	100:															// wait till password passes
		fbSoEWritePassword.Execute			:= FALSE;
		IF NOT fbSoEWritePassword.Busy THEN
			IF NOT fbSoEWritePassword.Error THEN
				iStep							:= iStep + 10;
			ELSE 
				udiADSerrorID					:= fbSoEWritePassword.AdsErrId;
				uiSoEErrorID					:= fbSoEWritePassword.SercosErrId;
				iLastStep						:= iStep;
				iStep							:= 999;
			END_IF
		END_IF
		
	110:															// Ignore offset error (P-0-0278), channel 1	
		P_0_0278_Value						:= 1;
		fbSoEWrite_ByDriveRef.stDriveRef	:= stDriveRef;
		fbSoEWrite_ByDriveRef.stDriveRef.nDriveNo:= 0;
		fbSoEWrite_ByDriveRef.nIdn			:= P_0_IDN  + 278;		// SoE Parameters Group P-0-IDN offset
		fbSoEWrite_ByDriveRef.nElement		:= EC_SOE_ELEMENT_VALUE;// Change value of the parameter
		fbSoEWrite_ByDriveRef.pSrcBuf		:= ADR(P_0_0278_Value);
		fbSoEWrite_ByDriveRef.cbBufLen		:= SIZEOF(P_0_0278_Value);
		fbSoEWrite_ByDriveRef.bExecute		:= TRUE;
		iStep								:= iStep + 10;				
		
	120,160:														// Writing done ?		
		fbSoEWrite_ByDriveRef.bExecute		:= FALSE;
		IF NOT fbSoEWrite_ByDriveRef.bBusy THEN
			IF NOT fbSoEWrite_ByDriveRef.bError THEN
				iStep							:= iStep + 10;
			ELSE
				udiADSerrorID					:= fbSoEWrite_ByDriveRef.iAdsErrId;
				uiSoEErrorID					:= fbSoEWrite_ByDriveRef.iSercosErrId;
				iLastStep						:= iStep;
				iStep							:= 999;
			END_IF	
		END_IF
		
	130:															// reset second channel if needed
		fbSoERead_ByDriveRef.stDriveRef		:= stDriveRef;
		fbSoERead_ByDriveRef.nIdn			:= P_0_IDN  + 324;		// SoE Parameters Group P-0-IDN offset
		fbSoERead_ByDriveRef.nElement		:= EC_SOE_ELEMENT_VALUE;// Change value of the parameter
		fbSoERead_ByDriveRef.pDstBuf		:= ADR(stSoE_String);
		fbSoERead_ByDriveRef.cbBufLen		:= SIZEOF(stSoE_String);
		fbSoERead_ByDriveRef.bExecute		:= TRUE;
		iStep								:= iStep + 10;				
		
	140:															// Reading done ?	skip reseting channel 2 for AX51xx	
		fbSoERead_ByDriveRef.bExecute		:= FALSE;
		IF NOT fbSoERead_ByDriveRef.bBusy THEN
			IF NOT fbSoERead_ByDriveRef.bError THEN
				bDualChannel := STRING_TO_BYTE(MID(stSoE_String.strData, 1, 4)) = 2;		// Sprawdza nazwe AX5xxx i rozpoznaje ilosc kanalow
				IF bDualChannel THEN
					iStep						:= iStep + 10;			// reset channel 2
				ELSE
					iStep						:= iStep + 30;			// skip reseting channel 2
				END_IF
			ELSE
				udiADSerrorID					:= fbSoERead_ByDriveRef.iAdsErrId;
				uiSoEErrorID					:= fbSoERead_ByDriveRef.iSercosErrId;
				iLastStep						:= iStep;
				iStep							:= 999;
			END_IF	
		END_IF
		
	150:															// Ignore offset error (P-0-0278), channel 2
		fbSoEWrite_ByDriveRef.stDriveRef.nDriveNo:= 1;
		fbSoEWrite_ByDriveRef.bExecute		:= TRUE;
		iStep								:= iStep + 10;

	170:															// Reset Drive (S-0-0099)
		fbSoEReset.Execute					:= TRUE; 
		fbSoEReset.NetId					:= ''; 
		iStep								:= iStep + 10;
		
	180:															// Wait for drive reset (S-0-0099)
		fbSoEReset.Execute					:= FALSE;
		IF NOT fbSoEReset.Busy THEN
			IF NOT fbSoEReset.Error THEN
				iStep							:= iStep + 10;
			ELSE
				udiADSerrorID					:= fbSoEReset.AdsErrId;
				uiSoEErrorID					:= fbSoEReset.SercosErrId;
				iLastStep						:= iStep;
				iStep							:= 999;
			END_IF
		END_IF
		
	190:															// Request OP State
		fbChangeSlaveState.byReguestedState	:= EC_DEVICE_STATE_OP;
		fbChangeSlaveState.bExecute			:= TRUE;
		iStep								:= iStep+10;
	
	200:															// Wait till state changed
		fbChangeSlaveState.bExecute			:= FALSE;	
		IF NOT fbChangeSlaveState.bBusy THEN
			IF NOT fbChangeSlaveState.bError THEN
				iStep							:= iStep+10;
			ELSE
				udiErrorID						:= fbChangeSlaveState.udiErrorID;
				iLastStep						:= iStep;
				iStep 							:= 999;
			END_IF				
		END_IF
		
	210:															// Set new encoder offset	
		fbSoEAX5000SetPositionOffset.Feedback:= ePositionOffsetFeedback1;	// set to feedback 1 only
		fbSoEAX5000SetPositionOffset.Execute:= TRUE; 
		iStep								:= iStep + 10;

	220:															//	offset set already?
		fbSoEAX5000SetPositionOffset.Execute:= FALSE;
		IF NOT fbSoEAX5000SetPositionOffset.Busy THEN
			IF NOT fbSoEAX5000SetPositionOffset.Error THEN
				iStep							:= iStep + 10;
			ELSE
				udiErrorID						:= fbSoEAX5000SetPositionOffset.ErrorID;
				iLastStep						:= iStep;
				iStep							:= 999;
			END_IF
		END_IF
	
	230:															//	FB Termination
		bBusy								:= FALSE;
		iStep								:= 0;

	999:															//	ERROR State
		bBusy								:=	FALSE;
		bError								:=	TRUE;
		iStep								:=	0;
	
END_CASE

fbAdsRead();
fbChangeSlaveState();
fbSoEWritePassword(Axis:=Axis);
fbSoEAX5000SetPositionOffset(Axis:=Axis);
fbSoEReadDiagNumber(Axis:=Axis);
fbSoEReset(Axis:=Axis);
fbSoEWrite_ByDriveRef();
fbSoERead_ByDriveRef();

END_FUNCTION_BLOCK

// ---- POUs/POUsAxisOnline/AX5000/FB_ChangeEtherCATSlaveState.TcPOU
//==================================================================================================
//							Beckhoff Automation Poland
//									23.05.2018
//	Blok zmienia stan EtherCAT Slave i monitoruje flage ukonczenia
//
//	Niezbedne biblioteki: Tc2_EtherCAT
//
// 	v1.1	|| TC v 3.1.4022.16	|| - optymalizacja kodu
// 	v1.0	|| TC v 3.1.4020.32	|| - pierwsza wersja
//==================================================================================================
FUNCTION_BLOCK FB_ChangeEtherCATSlaveState
VAR_INPUT
	bExecute								: BOOL;							// Start on rising edge
	sEtherCAT_NetID							: STRING;						// EtherCAT Master NetID
	nSlaveAddr								: UINT;							// EtherCAT Drive slave port
	byReguestedState						: BYTE;							(* 	16#1- EC_DEVICE_STATE_INIT  
																				16#2- EC_DEVICE_STATE_PREOP     
																				16#3- EC_DEVICE_STATE_BOOTSTRAP     
																				16#4- EC_DEVICE_STATE_SAFEOP  
																				16#8- EC_DEVICE_STATE_OP
																				16#10- EC_DEVICE_STATE_ERROR  *)
END_VAR
VAR_OUTPUT
	byActualState							: BYTE;							(* 	16#1-EC_DEVICE_STATE_INIT  
																				16#2-EC_DEVICE_STATE_PREOP     
																				16#3-EC_DEVICE_STATE_BOOTSTRAP     
																				16#4-EC_DEVICE_STATE_SAFEOP  
																				16#8-EC_DEVICE_STATE_OP
																				16#10-EC_DEVICE_STATE_ERROR  *)
	bBusy									: BOOL;
	bDone									: BOOL;
	bError									: BOOL;
	udiErrorID								: UDINT;	
END_VAR
VAR	
	fbEcReqSlaveState						: FB_EcReqSlaveState;
	fbEcGetSlaveState						: FB_EcGetSlaveState;
	timerTON								: TON;
	rtExecute								: R_TRIG;
	iState									: INT;
	iTry									: INT;							// number of tries
END_VAR

timerTON(PT:=T#500MS);
rtExecute(CLK:=bExecute);

CASE iState OF

	0:																// Init parameters
		IF rtExecute.Q THEN
			bBusy							:= TRUE;
			bDone							:= FALSE;
			bError							:= FALSE;
			udiErrorID						:= 0;
			iTry							:= 0;
			fbEcReqSlaveState.sNetId		:= sEtherCAT_NetID; 
			fbEcGetSlaveState.sNetId		:= sEtherCAT_NetID; 
			fbEcReqSlaveState.nSlaveAddr	:= nSlaveAddr; 
			fbEcGetSlaveState.nSlaveAddr	:= nSlaveAddr;
			fbEcReqSlaveState.state			:= byReguestedState;
			fbEcReqSlaveState.bExecute		:= TRUE;
			iState							:= iState + 10;			
		END_IF
		
	10:																// State request
		fbEcReqSlaveState.bExecute			:= FALSE;
		IF NOT fbEcReqSlaveState.bBusy THEN
			IF fbEcReqSlaveState.bError THEN
				iState						:= 99;
			ELSE
				iState						:= iState + 10;
			END_IF
		END_IF

		
	20:																// Request every 0.5s
		timerTON.IN							:= TRUE;
		IF timerTON.Q THEN
			timerTON.IN						:= FALSE;
			fbEcGetSlaveState.bExecute		:= TRUE;
			iState							:= iState + 10;
		END_IF
		
	30:																// Done already?
		fbEcGetSlaveState.bExecute			:= FALSE;	
		IF NOT fbEcGetSlaveState.bBusy THEN
			IF NOT fbEcGetSlaveState.bError AND fbEcGetSlaveState.state.deviceState = fbEcReqSlaveState.state THEN
				bBusy						:= FALSE;
				bDone						:= TRUE;
				iState						:= 0;
			ELSIF iTry = 40 THEN
				iState						:= 99;
			ELSE
				iTry						:= iTry + 1;
				iState						:= iState - 10;			
			END_IF
			byActualState					:= fbEcGetSlaveState.state.deviceState;
		END_IF
		
	99:																// ERROR STATE
		bError 								:= TRUE;
		bBusy								:= FALSE;
		udiErrorID							:= fbEcReqSlaveState.nErrId + fbEcGetSlaveState.nErrId;
		iState								:= 0;
		
END_CASE

fbEcReqSlaveState();
fbEcGetSlaveState();

END_FUNCTION_BLOCK

// ---- POUs/POUsAxisOnline/AX5000/FB_MotorMonitoringAX5000.TcPOU
//==================================================================================================
//							Beckhoff Automation Poland
//									22.09.2020
//	Blok funkcyjny pozwala na monitorowanie i ograniczanie momentu oraz monitoring parametru I2T dla AX5xxx.
//	Zmienne do zlinkowania zadeklarowane są wewnątrz bloku.
//	Ograniczenie i monitorowanie momentu
//	Ograniczenie momentu podawane jest przez wejście rTorqueLimit.
//	Na wyjściu podana jest wartość surowa w %, jak i przeskalowana na A (prąd) i Nm (moment).
//	Blok zwraca wartości bieżące, przefiltrowane i maksymalne.
//	Wartości maksymalne mogą być wyzerowane za pomocą zmiennej bReset.
//	Wewnętrznie wykorzystany jest blok FB_FilterEx.
//	I2T: 	Określamy okno czasowe pomiaru
//	Biblioteki: Tc2_MC2, Tc2_MC2_Drive, Tc2_Drive, Tc2_EtherCAT
//
// 	v1.4	|| TC v 3.1.4024.10		|| dostosowany do FW 2.13
// 	v1.3	|| TC v 3.1.4022.22		|| optymalizacja kod poprawiony blad wyliczenia Torque filtered
// 	v1.2	|| TC v 3.1.4022.22		|| optymalizacja kodu
// 	v1.1	|| TC v 3.1.4022.16		|| optymalizacja kodu, poprawiona flaga initialized
//  v1.0	|| TC v 3.1.4022.16		|| bazuje na FB_TorqueMonitoringEx2, dodane wyjscia zgodne z blokiem do AX8000 
//==================================================================================================
FUNCTION_BLOCK FB_MotorMonitoringAX5000
VAR CONSTANT
	rTorqueLimitLow					: REAL 		:= 0.01;				// Low limit used for bipolar torque limit value
	rTorqueLimitHigh				: REAL		:= 100.0;				// High limit used for bipolar torque limit value
END_VAR
VAR_INPUT
	bReset							: BOOL;
	rTorqueLimit					: REAL 		:= rTorqueLimitHigh; 	// Bipolar torque limit: 0-500%, resolution 0.1%, value goes to: 16#6072 (Ch A)/ 16#6872 (Ch B)
	tI2T_Window						: TIME 		:= T#100S;				// Has to be Task time * 100 * x 
																		// x - how many probes per measurement
																		// Samples - Task: 2 ms - tI2T_Window min 200 ms (1 probe), 100 probes then 20 s
																		// Task: 10 ms - tI2T_Window min 1 s (1 probe), 100 probes then 100 s
																		// If not proper time entered then it'll be adjusted
END_VAR
VAR_OUTPUT
	bError							: BOOL; 							// Communication error
	uiAdsErrId						: UINT;								// Forwarded output FB_SoeRead
	uiSercosErrId					: UINT;								// Forwarded output FB_SoeRead
	bInitialized					: BOOL;								// TRUE - Motor data read without errors, so it's possible to calculate torqe and current values in metric units
	bWarning						: BOOL;								// Overcurrent (rCurrentF > rRatedCurrent)
	rWarningCurrent					: REAL; 							// P_0_0093_Value in [A]
	rTorquePerc						: REAL;								// [%]
	rTorquePercMax					: REAL;								// Max [%]	
	rTorque							: REAL; 							// [Nm]
	rTorqueF						: REAL;								// Filtered
	rTorqueMax						: REAL;								// Max
	rCurrent						: REAL; 							// [A]
	rCurrentF						: REAL;								// Filtered
	rCurrentMax						: REAL;								// Max
	rI2T							: REAL; 							// % nominal
	rI2TMax							: REAL;
END_VAR
VAR_IN_OUT
	Axis							: AXIS_REF;
END_VAR
VAR
//======================== Internal =============================
	rTorqueRAW						: REAL; 							// -1000 .. 1000 - RAW values the same as process image	
	rContinuousStallTorque			: REAL; 							// P_0_0070_Value [Nm]
	rContinuousStallCurrent			: REAL; 							// S_0_0111_Value [A]
	rPeakCurrent					: REAL; 							// P_0_0092_Value in [A]
	rSfTorque						: REAL; 							// A --> Nm P_0_0070_Value/S_0_0111_Value [Nm/A]
	rSfCurrent						: REAL; 							// RAW --> A (-1000..1000 --> - rPeakCurrent .. rPeakCurrent)
	bFirstCycle						: BOOL := TRUE;
	iFW_High						: INT;
	iFW_Low							: INT;
	bDriveFirmware_GE_2_10			: BOOL;								// From FW >= 2.10 - different image size
	iFWPos							: INT;
	iFWLen							: INT;
	sDriveFW						: STRING(66);
	uiBipolarTorqueLimitValue AT %Q*	: UINT; 						// Raw data, linked to Bipolar torque limit value MDT, S-0-0092
	iStep							: INT;
	wInitErrorCount					: WORD;								// Initialization error counter, if bigger then 10 then error
	arr_S_0_0030_Value				: ARRAY [1..66] OF BYTE;			// till FW 2.10 total len is 66 bytes (2 - Act len, 2 - Max len, 62 - String 
	S_0_0030_Value					: STRING(61);
	P_0_0092_Value					: DWORD;
	P_0_0093_Value					: DWORD;
	P_0_0070_Value					: DWORD;
	S_0_0111_Value					: DWORD;
//========================== I2T ================================
	bCalculateI2T					: BOOL;								// TRUE in cycle when recalculation I2T necessary
	bBufferFull						: BOOL;								// TRUE when array buffer is full
	BIndex							: BYTE;								// Task no
	tI2T_WindowOld					: TIME;								// Old time window to reinit I2T calculation if necessary
	wProbeCyclesCount				: WORD;								// No of cycles for one I2T probe
	wCyclesCount					: WORD;								// Act no of cycles for one I2T probe
	wNoOfCycles						: WORD;								// Total cycles count for I2T window
	wNoOfProbes						: WORD;								// Actual number of probes for I2T calculation
	i								: INT;								// FOR loop
	rCycleTime						: REAL;								// Task time in [ms]
	rI2T_Window						: REAL;								// Time window in [ms]
	rCurrentPom						: REAL;								// Sum of current values in probe
	rCurrentAverage					: REAL;								// Arithmetical average
	rI2T_Nominal					: REAL;								// I2T for In
	rI2T_Actual						: REAL;								// I2T for real values
	arrI2TBuffer					: ARRAY[1..100] OF REAL;			// Buffer window to calculate I2T
//========================== FBs ================================
	rtReset							: R_TRIG;							// Reset trigger
	tonWait							: TON;								// Wait timer
	fbFilterEx						: FB_FilterEx;						// Filter
	fbSoERead						: FB_SoeRead;						// FB for read SoE parameters
	fbGETCURTASKINDEX   			: GETCURTASKINDEX;					// FB to check task no
//===============================================================
END_VAR

//===== Initialization, reinitialization and reset  =============
ACT_Init_Reset();
//=================== Call triggers and timers ==================
tonWait(IN:= NOT tonWait.Q, PT:= T#1S);
//============= Read params and calculations ====================
CASE iStep OF

	0: 	// Read S_0_0030 - Manufacturer version

		fbSoERead.Idn 					:= S_0_IDN + 30;
		fbSoERead.Element				:= EC_SOE_ELEMENT_VALUE;
		fbSoERead.pDstBuf				:= ADR(arr_S_0_0030_Value);
		fbSoERead.BufLen				:= SIZEOF(arr_S_0_0030_Value);
		fbSoERead.Execute				:= TRUE;
		iStep 							:= iStep + 10;

	10: // Wait till read finish 

		IF NOT fbSoERead.Busy THEN
			fbSoERead.Execute			:= FALSE;
			IF fbSoERead.Error THEN
				wInitErrorCount 		:= wInitErrorCount + 1;
				// Count > 10 then go to error and wait for reset, if not wait in warning step
				IF wInitErrorCount > 10 THEN
					uiAdsErrId			:= fbSoERead.AdsErrId;
					uiSercosErrId		:= fbSoERead.SercosErrId;
					iStep				:= 1000;								// Error step
				ELSE
					iStep				:= 900;									// Warning step
				END_IF
			ELSE
				iStep 					:= iStep + 5;
			END_IF
		END_IF

	15: // Read Drive firmware version

		MEMCPY(ADR(S_0_0030_Value), (ADR(arr_S_0_0030_Value)+4), 62);
		iFWPos							:= FIND(S_0_0030_Value,': v') + 3;
		sDriveFW						:= DELETE(S_0_0030_Value, iFWPos -1,1);
		iFWLen							:= FIND(sDriveFW,'.');
		iFW_High						:= STRING_TO_INT(LEFT(sDriveFW, iFWLen-1));
		sDriveFW						:= DELETE(sDriveFW,iFWLen,1);
		iFWLen							:= FIND(sDriveFW,' ');
		iFW_Low							:= STRING_TO_INT(LEFT(sDriveFW, iFWLen-1));
		
		bDriveFirmware_GE_2_10 			:= iFW_High >= 2 AND iFW_Low >= 10;				// Check if firmware >= 2.10
		iStep	 						:= iStep + 5;		

	20: // Read P_0_0092 - Configured channel peak current

		fbSoERead.Idn 					:= P_0_IDN + 92;
		fbSoERead.Element				:= EC_SOE_ELEMENT_VALUE;
		fbSoERead.pDstBuf				:= ADR(P_0_0092_Value);
		fbSoERead.BufLen				:= SIZEOF(P_0_0092_Value);
		fbSoERead.Execute				:= TRUE;
		iStep 							:= iStep + 10;

	30: // Wait till read finish 

		IF NOT fbSoERead.Busy THEN
			fbSoERead.Execute			:= FALSE;
			IF fbSoERead.Error THEN
				wInitErrorCount 		:= wInitErrorCount + 1;
				// Count > 10 then go to error and wait for reset, if not wait in warning step
				IF wInitErrorCount > 10 THEN
					uiAdsErrId			:= fbSoERead.AdsErrId;
					uiSercosErrId		:= fbSoERead.SercosErrId;
					iStep				:= 1000;								// Error step
				ELSE
					iStep				:= 900;									// Warning step
				END_IF
			ELSE
				iStep 					:= iStep + 10;
			END_IF
		END_IF

	40: // Read P_0_0070 - Motor continuous stall torque

		fbSoERead.Idn 					:= P_0_IDN + 70;
		fbSoERead.Element				:= EC_SOE_ELEMENT_VALUE; 
		fbSoERead.pDstBuf				:= ADR(P_0_0070_Value);
		fbSoERead.BufLen 				:= SEL(bDriveFirmware_GE_2_10, 2, 4);		// In FW GE 2.10 size is 4
		fbSoERead.Execute				:= TRUE;
		iStep 							:= iStep + 10;

	50: // Wait till read finish 

		IF NOT fbSoERead.Busy THEN
			fbSoERead.Execute			:= FALSE;
			IF fbSoERead.Error OR P_0_0070_Value = 0 THEN						// P_0_0070_Value = 0 - probably linear motor or wrong motor data
				wInitErrorCount 		:= wInitErrorCount + 1;
				// Count > 10 then go to error and wait for reset, if not wait in warning step
				IF wInitErrorCount > 10 THEN
					uiAdsErrId			:= fbSoERead.AdsErrId;
					uiSercosErrId		:= fbSoERead.SercosErrId;
					iStep				:= 1000;								// Error step
				ELSE
					iStep				:= 900;									// Warning step
				END_IF
			ELSE
				iStep 					:= iStep + 10;
			END_IF
		END_IF

	60: // Read S_0_0111 - Motor continuous stall current

		fbSoERead.Idn 					:= S_0_IDN + 111;
		fbSoERead.Element				:= EC_SOE_ELEMENT_VALUE;
		fbSoERead.pDstBuf				:= ADR(S_0_0111_Value);
		fbSoERead.BufLen				:= SIZEOF(S_0_0111_Value);
		fbSoERead.Execute				:= TRUE;
		iStep 							:= iStep + 10;
		
	70: // Wait till read finish 

		IF NOT fbSoERead.Busy THEN
			fbSoERead.Execute			:= FALSE;
			IF fbSoERead.Error OR S_0_0111_Value = 0 THEN			// S_0_0111_Value = 0 - wrong motor data
				wInitErrorCount 		:= wInitErrorCount + 1;
				// Count > 10 then go to error and wait for reset, if not wait in warning step
				IF wInitErrorCount > 10 THEN
					uiAdsErrId			:= fbSoERead.AdsErrId;
					uiSercosErrId		:= fbSoERead.SercosErrId;
					iStep				:= 1000;								// Error step
				ELSE
					iStep				:= 900;									// Warning step
				END_IF
			ELSE
				iStep 					:= iStep + 10;
			END_IF
		END_IF

	80: // Read P_0_0093 - Configured channel current

		fbSoERead.Idn 					:= P_0_IDN + 93;
		fbSoERead.Element				:= EC_SOE_ELEMENT_VALUE;
		fbSoERead.pDstBuf				:= ADR(P_0_0093_Value);
		fbSoERead.BufLen				:= SIZEOF(P_0_0093_Value);
		fbSoERead.Execute				:= TRUE;
		iStep 							:= iStep + 10;
	
	90: // Wait till read finish 

		IF NOT fbSoERead.Busy THEN
			fbSoERead.Execute			:= FALSE;
			IF fbSoERead.Error THEN
				wInitErrorCount 		:= wInitErrorCount + 1;
				// Count > 10 then go to error and wait for reset, if not wait in warning step
				IF wInitErrorCount > 10 THEN
					uiAdsErrId			:= fbSoERead.AdsErrId;
					uiSercosErrId		:= fbSoERead.SercosErrId;
					iStep				:= 1000;								// Error step
				ELSE
					iStep				:= 900;									// Warning step
				END_IF
			ELSE
				iStep 					:= iStep + 10;							
			END_IF
		END_IF
		
	100: // Read data from unit finished - we can calculate params

		rPeakCurrent 					:= DWORD_TO_REAL(P_0_0092_Value) / 1000.0;		// In [A]
		rSfCurrent 						:= rPeakCurrent / 1000.0;						// iTorque -1000..1000 --> - rPeakCurrent .. rPeakCurrent
		rContinuousStallTorque 			:= DWORD_TO_REAL(P_0_0070_Value) / 100;
		rContinuousStallCurrent 		:= DWORD_TO_REAL(S_0_0111_Value) / 1000;
		IF rContinuousStallCurrent <> 0 THEN
			rSfTorque	 				:= rContinuousStallTorque / rContinuousStallCurrent;
		END_IF
		rWarningCurrent 				:= DWORD_TO_REAL(P_0_0093_Value) / 1000;
		iStep 							:= 200;

	200: // Read cycle time - we need it for I2T calculations

		fbGETCURTASKINDEX(index => BIndex);
		IF BIndex <> 0 THEN
			iStep						:= iStep + 10;
		END_IF

	210:

		rCycleTime 						:= UDINT_TO_REAL(_TaskInfo[BIndex].CycleTime) / 10000.0;	// Scale to [ms]
		rI2T_Window 					:= TIME_TO_REAL(tI2T_Window);
		wNoOfCycles						:= REAL_TO_WORD(rI2T_Window / rCycleTime);
		// Time window too short
		IF wNoOfCycles < 100 THEN
			iStep						:= 1000;								// Error step
		ELSE
			wProbeCyclesCount 			:= wNoOfCycles / 100;
			iStep						:= 300;
		END_IF

	300: // Calculations	

		ACT_I2T();
	
	900: // Warning - wait and repeat read - problem during read motor data, i.e. EtherCAT doesn't work yet

		IF tonWait.Q THEN
			iStep 						:= 0;	// Repeat initialization phase 
		END_IF
		
	1000: // Error - wait for reset 
		;

END_CASE
//===============================================================

bError		 							:= iStep = 1000;
bInitialized 							:= iStep >= 300 AND NOT bError;
ACT_Calculations();

//========================= Warning =============================
bWarning								:= rCurrentF > rWarningCurrent;

//===================== Limit output torque =====================
IF rTorqueLimit < rTorqueLimitLow THEN
	uiBipolarTorqueLimitValue 			:= REAL_TO_UINT(rTorqueLimitHigh);			// Secure against 0 value - probably empty var connected to input
ELSE
	uiBipolarTorqueLimitValue 			:= REAL_TO_UINT(LIMIT(rTorqueLimitLow,rTorqueLimit,rTorqueLimitHigh)) * 10;
END_IF

//====================== Call SoE read FB =======================
fbSoERead(	NetId:= '',
			Timeout:= T#1s,
			Axis:= Axis);

ACTION ACT_Calculations:
//============== Raw values - always avaliable ==================
rTorquePerc								:= LREAL_TO_REAL(Axis.NcToPlc.ActTorque); 		// [%]
rTorqueRAW 								:= rTorquePerc * 10;							// -1000 .. 1000 - RAW values the same as process image
//===================== Filter current value ====================
fbFilterEx(rIn:= rTorqueRAW, tTimeConstant:= T#1S);

// Calculations	- possible only with params
IF bInitialized THEN
	rCurrent 							:= rTorqueRAW * rSfCurrent;
	rTorque 							:= rCurrent * rSfTorque;
	rCurrentF 							:= fbFilterEx.rOut * rSfCurrent;
	rTorqueF 							:= rCurrentF * rSfTorque;
END_IF

//=============== Save torque and current max values ===============
IF ABS(rCurrentMax) < ABS(rCurrentF) THEN
	rTorquePercMax						:= rTorquePerc;
	rCurrentMax 						:= rCurrentF;
	rTorqueMax 							:= rTorqueF;
END_IF
END_ACTION

ACTION ACT_I2T:
//======================= One probe =============================
rCurrentPom 							:= rCurrentPom + ABS(rCurrent);
wCyclesCount							:= wCyclesCount + 1;
bCalculateI2T							:= FALSE;
IF wCyclesCount = wProbeCyclesCount THEN
	rCurrentAverage 					:= rCurrentPom / WORD_TO_REAL(wProbeCyclesCount);
	rCurrentPom							:= 0;
	wCyclesCount						:= 0;
	bCalculateI2T						:= TRUE;							
ELSIF wCyclesCount > wProbeCyclesCount THEN
	iStep 								:= 1000;
END_IF
//===============================================================

//==================== Recalculate I2T ==========================
IF bCalculateI2T THEN
	wNoOfProbes 						:= wNoOfProbes + 1;
	bBufferFull 						:= wNoOfProbes >= 100;
	MEMMOVE(ADR(arrI2TBuffer) + 4, ADR(arrI2TBuffer), SIZEOF(arrI2TBuffer) - 4);
	arrI2TBuffer[1]						:= rCurrentAverage;
	IF bBufferFull THEN
		rI2T_Nominal					:= 100.0 * rContinuousStallCurrent;
		rI2T_Actual						:= 0;
		FOR i := 1 TO 100 DO
			rI2T_Actual					:= rI2T_Actual + arrI2TBuffer[i];
		END_FOR
	ELSE
		rI2T_Nominal					:= wNoOfProbes * rContinuousStallCurrent;
		rI2T_Actual						:= rI2T_Actual + rCurrentAverage;
	END_IF
	rI2T								:= rI2T_Actual * 100 / rI2T_Nominal; // In [%]
//====================== Save I2T max value =====================
	IF rI2TMax < rI2T THEN
		rI2TMax							:= rI2T;
	END_IF
END_IF
//===============================================================
END_ACTION

ACTION ACT_Init_Reset:
//============== Reset max values and FB ========================
rtReset(CLK:= bReset);
// Reset I2T calculations when time window changed or reset CMD
IF rtReset.Q OR tI2T_Window <> tI2T_WindowOld THEN
	BIndex								:= 0;
	wProbeCyclesCount					:= 0;
	wCyclesCount						:= 0;
	wNoOfCycles							:= 0;
	wNoOfProbes							:= 0;
	i									:= 0;
	rCycleTime							:= 0;
	rI2T_Window							:= 0;
	rCurrentPom							:= 0;
	rCurrentAverage						:= 0;
	rI2T_Nominal						:= 0;
	rI2T_Actual							:= 0;
	rI2T								:= 0;
	rI2TMax								:= 0;
	MEMSET(ADR(arrI2TBuffer), 0, SIZEOF(arrI2TBuffer));
	bBufferFull							:= FALSE;
	bCalculateI2T						:= FALSE;
	// If there is no Error then recalculate time-dipendent variables
	IF NOT bError THEN
		iStep							:= 200;
	END_IF
	tI2T_WindowOld 						:= tI2T_Window;
END_IF

IF rtReset.Q OR bFirstCycle THEN
	fbSoERead.Execute					:= FALSE;
	bWarning	 						:= FALSE;
	bDriveFirmware_GE_2_10 				:= FALSE;
	uiAdsErrId		 					:= 0;
	uiSercosErrId	 					:= 0;
	rWarningCurrent 					:= 0;
	rTorquePerc 						:= 0;
	rTorquePercMax 						:= 0;
	rTorque 							:= 0;
	rTorqueF 							:= 0;
	rTorqueMax 							:= 0;
	rCurrent 							:= 0;
	rCurrentF 							:= 0;
	rCurrentMax 						:= 0;
	rTorqueRAW 							:= 0;
	rContinuousStallTorque 				:= 0;
	rContinuousStallCurrent 			:= 0;
	rPeakCurrent 						:= 0;
	rSfTorque 							:= 0;
	rSfCurrent							:= 0;
	iStep								:= 0;
	wInitErrorCount						:= 0;
	MEMSET(ADR(arr_S_0_0030_Value), 0, SIZEOF(arr_S_0_0030_Value));
	S_0_0030_Value						:= '';
	P_0_0092_Value						:= 0;
	P_0_0093_Value						:= 0;
	P_0_0070_Value						:= 0;
	S_0_0111_Value						:= 0;
	bFirstCycle	 						:= FALSE;
END_IF
END_ACTION

END_FUNCTION_BLOCK

// ---- POUs/POUsAxisOnline/AX5000/FB_AxisDiag.TcPOU
//==================================================================================================
//							Beckhoff Automation Poland
//								23.05.2018
//					Blok do diagnostyki osi
// 	v1.1	|| TC v 3.1.4022.16	|| - optymalizacja kodu
// 	v1.0	|| TC v 3.1.4020.0	|| - pierwsza wersja
//==================================================================================================
FUNCTION_BLOCK FB_AxisDiag
VAR_INPUT
	IPCNetID							: T_AmsNetId; 	(* AmsNetId of the IPC *)
	Timeout								: TIME := DEFAULT_ADS_TIMEOUT;
	Reset								: BOOL;
	GetDiag								: BOOL;
END_VAR
VAR_IN_OUT
	Axis	 							: AXIS_REF;
	stAX5000Diag						: ST_AX5000Diag;
END_VAR
VAR_OUTPUT
	Error								: BOOL;
	AdsErrId							: UINT;
	SercosErrId							: UINT;
	ResetAct							: BOOL;
	DiagAct								: BOOL;
	Busy								: BOOL;
END_VAR
VAR
	iState								: INT;
	iSubState							: INT;
	GetDriveRef							: BOOL;
	DriveRef								: ST_DriveRef; (* contains sNetID of EcMaster, nSlaveAddr of EcDrive, nDriveNo of EcDrive, either preset or read from NC *)
	AxisID								: UDINT;

	C1DErrorPrev							: BOOL;
	WcStateErrorPrev						: BOOL;
	AxisErrorPrev							: BOOL;
	OperationalPrev						: BOOL;
	ResetPrev							: BOOL;
	GetDiagPrev							: BOOL;

	fbSoERead							: FB_SoERead;
	fbDiagMessage 						: FB_SoEReadDiagMessage;
	fbClassXDiag							: FB_SoEReadClassXDiag;
	fbDiagNumber						: FB_SoEReadDiagNumber;
	fbDiagNumberList						: FB_SoEReadDiagNumberList;

	fbReset								: FB_SoEReset;
	fbDelay								: TON;
	fbGetSlaveState 						: FB_EcGetSlaveState;
	fbReqSlaveState 						: FB_EcReqSlaveState;
	fbNcReset 							: MC_Reset;

	fbAdsRead							: ADSREAD;
	readBuffer							: ARRAY[0..9] OF BYTE;
	Ids									: T_AmsNetIdArr;
	strSoEString							: ST_SoE_String;
END_VAR
VAR CONSTANT
	NCIDXG_AXPARMS					: UDINT := 16#00004000;	(* Axis with ID: Parameter 			*)
	NCIDXO_AXP_HWAMSADDR			: UDINT := 16#00000031;
END_VAR

stAX5000Diag.bOperational	:= Axis.NcToPlc.StateDWord.0;
stAX5000Diag.bC1DError	 	:= Axis.NcToPlc.StateDWord.28;
stAX5000Diag.bWcStateError 	:= Axis.NcToPlc.StateDWord.30;
stAX5000Diag.bAxisError		:= Axis.NcToPlc.StateDWord.31;
stAX5000Diag.iAxisErrorCode	:= Axis.NcToPlc.ErrorCode;

CASE iState OF
0:	(* idle *)
	GetDriveRef 	:= (DriveRef.nSlaveAddr = 0);

	IF GetDriveRef THEN
		Busy			:= TRUE;
		Error			:= FALSE;
		AdsErrId		:= 0;
		SercosErrId		:= 0;
		iState 			:= 1;
		iSubState		:= 0;
		AxisID 			:= Axis.NcToPlc.AxisId;

	ELSIF Reset AND NOT ResetPrev THEN
		Busy			:= TRUE;
		ResetAct		:= TRUE;
		ResetPrev		:= Reset;
		Error			:= FALSE;
		AdsErrId		:= 0;
		SercosErrId		:= 0;
		iState 			:= 2;
		iSubState		:= 0;
		AxisID 			:= Axis.NcToPlc.AxisId;

	ELSIF GetDiag AND NOT GetDiagPrev OR
		(stAX5000Diag.bC1DError AND NOT C1DErrorPrev) OR (NOT stAX5000Diag.bC1DError AND C1DErrorPrev) (* rising/falling C1D *) OR
		(stAX5000Diag.bWcStateError AND NOT WcStateErrorPrev) OR (NOT stAX5000Diag.bWcStateError AND WcStateErrorPrev) (* rising/falling WcState *) OR
		(stAX5000Diag.bAxisError AND NOT AxisErrorPrev) OR (NOT stAX5000Diag.bAxisError AND AxisErrorPrev) (* rising/falling NcError *) OR
		(stAX5000Diag.bOperational AND NOT OperationalPrev) OR (NOT stAX5000Diag.bOperational AND OperationalPrev) (* rising/falling Enable *) THEN

		Busy			:= TRUE;
		DiagAct			:= TRUE;
		GetDiagPrev		:= GetDiag;
		Error			:= FALSE;
		AdsErrId		:= 0;
		SercosErrId		:= 0;
		iState 			:= 3;
		iSubState		:= 0;
		AxisID 			:= Axis.NcToPlc.AxisId;

		(* set/clear flags *)
		C1DErrorPrev		:= stAX5000Diag.bC1DError;
		WcStateErrorPrev	:= stAX5000Diag.bWcStateError;
		AxisErrorPrev		:= stAX5000Diag.bAxisError;
		OperationalPrev		:= stAX5000Diag.bOperational;

	ELSE
		ResetAct	:= FALSE;
		DiagAct		:= FALSE;
	END_IF

1:	(* get drive reference *)
	M_GetDriveRef();

2:	(* reset and state change *)
	M_Reset();

3:	(* get diag data *)
	M_GetDiagnosis();

END_CASE

(* clear latch *)
ResetPrev	:= ResetPrev AND Reset;
GetDiagPrev	:= GetDiagPrev AND GetDiag;

ACTION M_GetDiagnosis:
CASE iSubState OF
0:	fbClassXDiag(
		NetId		:= IPCNetID,
		Execute		:= TRUE,
		DiagClass 	:= 1,
		Timeout		:= DEFAULT_ADS_TIMEOUT,
		Axis		:= Axis,
	);

	IF NOT fbClassXDiag.Busy THEN
		fbClassXDiag(Execute:= FALSE,Axis := Axis);

		IF NOT fbClassXDiag.Error THEN
			stAX5000Diag.wClass1Diag	:= fbClassXDiag.ClassXDiag;
			stAX5000Diag.stClass1Diag	:= F_ConvWordToSTAX5000C1D(stAX5000Diag.wClass1Diag);
		ELSE
			Error			:= TRUE;
			AdsErrId		:= fbClassXDiag.AdsErrId;
			SercosErrId	:= fbClassXDiag.SercosErrId;
		END_IF
		iSubState	:= iSubState + 1;
	END_IF

1:	fbDiagMessage(
		NetId	:= IPCNetID,
		Execute	:= TRUE,
		Timeout	:= DEFAULT_ADS_TIMEOUT,
		Axis	:= Axis,
	);

	IF NOT fbDiagMessage.Busy THEN
		fbDiagMessage(Execute:= FALSE,Axis := Axis);

		IF NOT fbDiagMessage.Error THEN
			stAX5000Diag.strDiagMessage := LEFT(fbDiagMessage.DiagMessage.strData, UINT_TO_INT(fbDiagMessage.DiagMessage.iActualSize));
		ELSE
			Error			:= TRUE;
			AdsErrId		:= fbDiagMessage.AdsErrId;
			SercosErrId	:= fbDiagMessage.SercosErrId;
		END_IF
		iSubState	:= iSubState + 1;
	END_IF

2:	fbDiagNumber(
		NetId	:= IPCNetID,
		Execute	:= TRUE,
		Timeout	:= DEFAULT_ADS_TIMEOUT,
		Axis	:= Axis,
	);

	IF NOT fbDiagNumber.Busy THEN
		fbDiagNumber(Execute:= FALSE,Axis := Axis);

		IF NOT fbDiagNumber.Error THEN
			stAX5000Diag.iDiagNumber := fbDiagNumber.DiagNumber;
		ELSE
			Error			:= TRUE;
			AdsErrId		:= fbDiagNumber.AdsErrId;
			SercosErrId	:= fbDiagNumber.SercosErrId;
		END_IF
		iSubState	:= iSubState + 1;
	END_IF

3:	fbSoERead(
		NetId	:= IPCNetID,
		Execute	:= TRUE,
		Idn		:= 135,
		Element	:=16#44,
		pDstBuf	:=ADR(stAX5000Diag.wDriveStatus),
		BufLen	:=SIZEOF(stAX5000Diag.wDriveStatus),
		Timeout	:= DEFAULT_ADS_TIMEOUT,
		Axis	:= Axis,
	);

	IF NOT fbSoERead.Busy THEN
		fbSoERead(Execute:= FALSE,Axis := Axis);
		IF NOT fbSoERead.Error THEN
			stAX5000Diag.stDriveStatus := F_ConvWordToSTAX5000DriveStatus(stAX5000Diag.wDriveStatus);
			iSubState		:= iSubState + 1;
		ELSE
			Error			:= TRUE;
			AdsErrId		:= fbSoERead.AdsErrId;
			SercosErrId	:= fbSoERead.SercosErrId;
			iSubState		:= iSubState + 2;
		END_IF
	END_IF

4:	fbSoERead(
		NetId	:= IPCNetID,
		Execute	:= TRUE,
		Idn		:= stAX5000Diag.stDriveStatus.iActOpModeParNum,
		Element	:=16#44,
		pDstBuf	:=ADR(stAX5000Diag.stDriveStatus.eActOpMode),
		BufLen	:=SIZEOF(stAX5000Diag.stDriveStatus.eActOpMode),
		Timeout	:= DEFAULT_ADS_TIMEOUT,
		Axis	:= Axis,
	);

	IF NOT fbSoERead.Busy THEN
		fbSoERead(Execute:= FALSE,Axis := Axis);
		IF NOT fbSoERead.Error THEN
			;
		ELSE
			Error			:= TRUE;
			AdsErrId		:= fbSoERead.AdsErrId;
			SercosErrId	:= fbSoERead.SercosErrId;
		END_IF
		iSubState	:= iSubState + 1;
	END_IF

5:	fbGetSlaveState(
		sNetId		:= DriveRef.sNetId,
		nSlaveAddr	:= DriveRef.nSlaveAddr,
		bExecute	:= TRUE,
		tTimeout	:= DEFAULT_ADS_TIMEOUT,
	);

	IF NOT fbGetSlaveState.bBusy THEN
		fbGetSlaveState(bExecute:= FALSE);
		IF NOT fbGetSlaveState.bError THEN
			stAX5000Diag.stEcSlaveState := fbGetSlaveState.state;
			stAX5000Diag.stEcSlaveStateBits := F_ConvSlaveStateToBits(fbGetSlaveState.state);
		ELSE
			Error			:= TRUE;
			AdsErrId		:= UDINT_TO_UINT(fbGetSlaveState.nErrId);
		END_IF

		IF stAX5000Diag.stEcSlaveStateBits.bError THEN
			IF stAX5000Diag.stEcSlaveStateBits.bPreop THEN
				(* read S21 - IDN List of Invalid operation data for CP2 (Preop->SaveOp) *)
				MEMSET(ADR(stAX5000Diag.stCPxInvParamList), 0, SIZEOF(stAX5000Diag.stCPxInvParamList));
				stAX5000Diag.bPreopToSafeOpError := TRUE;
				stAX5000Diag.bSafeOpToOpError := FALSE;
				iSubState	:= iSubState + 1;
			ELSIF stAX5000Diag.stEcSlaveStateBits.bSafeOp THEN
				(* read S22 - IDN List of Invalid operation data for CP3 (SaveOp->Op) *)
				MEMSET(ADR(stAX5000Diag.stCPxInvParamList), 0, SIZEOF(stAX5000Diag.stCPxInvParamList));
				stAX5000Diag.bPreopToSafeOpError := FALSE;
				stAX5000Diag.bSafeOpToOpError := TRUE;
				iSubState	:= iSubState + 2;
			ELSE
				(* Skip S21 + S22 *)
				MEMSET(ADR(stAX5000Diag.stCPxInvParamList), 0, SIZEOF(stAX5000Diag.stCPxInvParamList));
				stAX5000Diag.bPreopToSafeOpError := FALSE;
				stAX5000Diag.bSafeOpToOpError := FALSE;
				iSubState	:= iSubState + 3;
			END_IF
		ELSE
			(* Skip S21 + S22 *)
			MEMSET(ADR(stAX5000Diag.stCPxInvParamList), 0, SIZEOF(stAX5000Diag.stCPxInvParamList));
			stAX5000Diag.bPreopToSafeOpError := FALSE;
			stAX5000Diag.bSafeOpToOpError := FALSE;
			iSubState	:= iSubState + 3;
		END_IF
	END_IF

6:	(* read S21 - IDN List of Invalid operation data for CP2 (Preop->SaveOp) *)
	fbSoERead(
		NetId	:= IPCNetID,
		Execute	:= TRUE,
		Idn		:= 21,
		Element	:=16#40,
		pDstBuf	:=ADR(stAX5000Diag.stCPxInvParamList),
		BufLen	:=SIZEOF(stAX5000Diag.stCPxInvParamList),
		Timeout	:= DEFAULT_ADS_TIMEOUT,
		Axis	:= Axis,
	);

	IF NOT fbSoERead.Busy THEN
		fbSoERead(Execute:= FALSE,Axis := Axis);
		IF NOT fbSoERead.Error THEN
			;
		ELSE
			Error			:= TRUE;
			AdsErrId		:= fbSoERead.AdsErrId;
			SercosErrId	:= fbSoERead.SercosErrId;
		END_IF
		iSubState	:= iSubState + 2;
	END_IF

7:	(* read S22 - IDN List of Invalid operation data for CP3 (SaveOp->Op) *)
	fbSoERead(
		NetId	:= IPCNetID,
		Execute	:= TRUE,
		Idn		:= 22,
		Element	:=16#40,
		pDstBuf	:=ADR(stAX5000Diag.stCPxInvParamList),
		BufLen	:=SIZEOF(stAX5000Diag.stCPxInvParamList),
		Timeout	:= DEFAULT_ADS_TIMEOUT,
		Axis	:= Axis,
	);

	IF NOT fbSoERead.Busy THEN
		fbSoERead(Execute:= FALSE,Axis := Axis);
		IF NOT fbSoERead.Error THEN
			;
		ELSE
			Error			:= TRUE;
			AdsErrId		:= fbSoERead.AdsErrId;
			SercosErrId	:= fbSoERead.SercosErrId;
		END_IF
		iSubState	:= iSubState + 1;
	END_IF

8:	fbDiagNumberList(
		NetId			:= IPCNetID,
		Execute			:= TRUE,
		Timeout			:= DEFAULT_ADS_TIMEOUT,
		pDiagNumber		:= ADR(stAX5000Diag.stDiagNumberList),
		Size			:= SIZEOF(stAX5000Diag.stDiagNumberList),
		Axis			:= Axis,
	);

	IF NOT fbDiagNumberList.Busy THEN
		fbDiagNumberList(Execute:= FALSE,Axis := Axis);

		IF fbDiagNumberList.Error THEN
			Error			:= TRUE;
			AdsErrId		:= fbDiagNumberList.AdsErrId;
			SercosErrId	:= fbDiagNumberList.SercosErrId;
		END_IF

		IF (stAX5000Diag.strMotorType = '') OR (stAX5000Diag.strDriveType = '') THEN
			iSubState	:= iSubState + 1;
		ELSE
			DiagAct	:= FALSE;
			iSubState	:= 0;
			iState		:= 0;
			Busy		:= FALSE;
		END_IF
	END_IF

9:	fbSoERead(
		NetId	:= IPCNetID,
		Execute	:= TRUE,
		Idn		:= P_0_IDN + 53,
		Element	:=16#44,
		pDstBuf	:=ADR(strSoEString),
		BufLen	:=SIZEOF(strSoEString),
		Timeout	:= DEFAULT_ADS_TIMEOUT,
		Axis	:= Axis,
	);

	IF NOT fbSoERead.Busy THEN
		fbSoERead(Execute:= FALSE,Axis := Axis);
		IF NOT fbSoERead.Error THEN
			MEMSET(ADR(stAX5000Diag.strMotorType),0,SIZEOF(stAX5000Diag.strMotorType));
			MEMCPY(ADR(stAX5000Diag.strMotorType),ADR(strSoEString.strData),MIN(SIZEOF(stAX5000Diag.strMotorType),strSoEString.iActualSize));
		ELSE
			Error			:= TRUE;
			AdsErrId		:= fbSoERead.AdsErrId;
			SercosErrId	:= fbSoERead.SercosErrId;
		END_IF
		iSubState	:= iSubState + 1;
	END_IF

10:	fbSoERead(
		NetId	:= IPCNetID,
		Execute	:= TRUE,
		Idn		:= P_0_IDN + 324,
		Element	:=16#44,
		pDstBuf	:=ADR(strSoEString),
		BufLen	:=SIZEOF(strSoEString),
		Timeout	:= DEFAULT_ADS_TIMEOUT,
		Axis	:= Axis,
	);

	IF NOT fbSoERead.Busy THEN
		fbSoERead(Execute:= FALSE,Axis := Axis);
		IF NOT fbSoERead.Error THEN
			MEMSET(ADR(stAX5000Diag.strDriveType),0,SIZEOF(stAX5000Diag.strDriveType));
			MEMCPY(ADR(stAX5000Diag.strDriveType),ADR(strSoEString.strData),MIN(SIZEOF(stAX5000Diag.strDriveType),strSoEString.iActualSize));
		ELSE
			Error			:= TRUE;
			AdsErrId		:= fbSoERead.AdsErrId;
			SercosErrId	:= fbSoERead.SercosErrId;
		END_IF
		DiagAct	:= FALSE;
		iSubState	:= 0;
		iState		:= 0;
		Busy		:= FALSE;
	END_IF


END_CASE
END_ACTION

ACTION M_GetDriveRef:
(* get reference from NC *)
fbAdsRead(
	NETID	:= IPCNetID,
	PORT	:= AMSPORT_R0_NC,
	IDXGRP	:= NCIDXG_AXPARMS + Axis.NcToPlc.AxisId,
	IDXOFFS	:= NCIDXO_AXP_HWAMSADDR,
	LEN		:= SIZEOF(readBuffer) ,
	DESTADDR:= ADR(readBuffer),
	READ	:= TRUE,
	TMOUT	:= Timeout
);

IF NOT fbAdsRead.BUSY THEN
	fbAdsRead(READ := FALSE);
	stAX5000Diag.nNCAxisID := Axis.NcToPlc.AxisId;

	IF NOT fbAdsRead.ERR THEN
		MEMCPY(ADR(Ids), ADR(readBuffer), SIZEOF(Ids)); 										(* readBuffer[0..5] *)
		MEMCPY(ADR(DriveRef.nSlaveAddr), ADR(readBuffer[6]), SIZEOF(DriveRef.nSlaveAddr));  	(* readBuffer[6..7] *)
		MEMCPY(ADR(DriveRef.nDriveNo), ADR(readBuffer[8]), SIZEOF(DriveRef.nDriveNo));  		(* readBuffer[8..9] *)

		(* create string out of byte array *)
		DriveRef.sNetId := F_CreateAmsNetId(Ids);
		GetDriveRef := FALSE;
	END_IF

	Busy	:= FALSE;
	iState	:= 0;
END_IF
END_ACTION

ACTION M_Reset:
CASE iSubState OF
0:
	IF stAX5000Diag.bWcStateError OR stAX5000Diag.bC1DError THEN
		(* ResetAmplifier *)
		iSubState := iSubState + 1;
	ELSIF (NOT stAX5000Diag.bOperational) OR stAX5000Diag.bAxisError OR (stAX5000Diag.iAxisErrorCode <> 0) THEN
		(* NC Reset only *)
		iSubState := 6;
	ELSE
		(* reset not required *)
		iSubState	:= 0;
		iState		:= 0;
		Busy		:= FALSE;
		ResetAct	:= FALSE;
	END_IF

1:	(* ResetAmplifier *)
	fbReset(
		NetId	:= IPCNetID,
		Execute	:= TRUE,
		Timeout	:= DEFAULT_ADS_TIMEOUT,
		Axis	:= Axis,
	);
	IF NOT fbReset.Busy THEN
		fbReset(Execute:= FALSE, Axis:= Axis);

		IF NOT fbReset.Error THEN
			iSubState	:= iSubState + 1;
		ELSE
			Error			:= TRUE;
			AdsErrId		:= fbReset.AdsErrId;
			SercosErrId		:= fbReset.SercosErrId;
			Busy			:= FALSE;
			ResetAct		:= FALSE;
			iSubState		:= 0;
			iState			:= 0;
		END_IF
	END_IF

2:	fbDelay(IN:=TRUE, PT:=t#3s);
	IF fbDelay.Q THEN
		fbDelay(IN:=FALSE);
		iSubState	:= iSubState + 1;
	END_IF

3:	fbGetSlaveState(
		sNetId		:= DriveRef.sNetId,
		nSlaveAddr	:= DriveRef.nSlaveAddr,
		bExecute	:= TRUE,
		tTimeout	:= DEFAULT_ADS_TIMEOUT,
	);

	IF NOT fbGetSlaveState.bBusy THEN
		fbGetSlaveState(bExecute:= FALSE);

		IF NOT fbGetSlaveState.bError THEN
			IF Axis.NcToPlc.StateDWord.31 OR (Axis.NcToPlc.ErrorCode <> 0) THEN
				iSubState	:= 6;
			ELSE
				Busy		:= FALSE;
				ResetAct	:= FALSE;
				iSubState	:= 0;
				iState		:= 0;
			END_IF
		ELSE
			Error			:= TRUE;
			AdsErrId		:= UDINT_TO_UINT(fbGetSlaveState.nErrId);
			Busy			:= FALSE;
			ResetAct		:= FALSE;
			iSubState		:= 0;
			iState			:= 0;
		END_IF
	END_IF

5:	(* set op *)
	fbReqSlaveState(
		sNetId		:= DriveRef.sNetId,
		nSlaveAddr	:= DriveRef.nSlaveAddr,
		bExecute	:= TRUE,
		tTimeout	:= DEFAULT_ADS_TIMEOUT,
		state		:= EC_DEVICE_STATE_OP);

	IF NOT fbReqSlaveState.bBusy THEN
		fbReqSlaveState(bExecute:= FALSE);

		IF NOT fbReqSlaveState.bError THEN
			iSubState	:= iSubState + 1;
		ELSE
			Error		:= TRUE;
			AdsErrId	:= UDINT_TO_UINT(fbReqSlaveState.nErrId);
			Busy		:= FALSE;
			ResetAct	:= FALSE;
			iSubState	:= 0;
			iState		:= 0;
		END_IF
	END_IF

6:	fbNcReset(
		Execute:= TRUE,
		Axis:= Axis,
	);
	IF fbNcReset.Done OR fbNcReset.Error THEN
		IF fbNcReset.Error THEN
			Error 		:= TRUE;
			AdsErrId 	:= UDINT_TO_UINT(fbNcReset.ErrorID);
		END_IF

		iSubState	:= 0;
		iState		:= 0;
		Busy		:= FALSE;
		ResetAct	:= FALSE;
		fbNcReset(Execute:= FALSE, Axis:= Axis);
	END_IF
END_CASE
END_ACTION

END_FUNCTION_BLOCK

// ---- POUs/POUsAxisOnline/FBs/F_AxErrMsg.TcPOU
//==================================================================================================
//							Beckhoff Automation Poland
//								7.12.2018
//		Funkcja konwertujaca nr bledu na opis
// 	v1.0	|| TC v 3.1.4022.27	|| - pierwsza wersja
//==================================================================================================
FUNCTION F_AxErrMsg : STRING(255)
VAR_INPUT
	iErrID: UDINT;
END_VAR
VAR
	sMsg: STRING(255);
END_VAR

(* these err msgs are taken straight from infosys ....
http://infosys.beckhoff.com/content/1033/tcncerrcode/html/tcncerrorcodesoverview.htm?id=27430  
*)

IF iErrID < 1 THEN
	sMsg := '';
	F_AxErrMsg := sMsg;
	RETURN;
END_IF

CASE iErrID OF
(* NC AXIS ERRORS *)
	16#4000: sMsg := '4000 internal "Internal error" Internal system error in the NC on ring 0, no further details.';
	16#4001: sMsg := '4001 memory "Memory error" The ring-0 memory management is not providing the required memory. This is usually a result of another error, as a result of which the controller will halt normal operation (now if not …';
	16#4002: sMsg := '4002 internal "Nc retain data error (persistent data)" Error while loading the Nc retain data. The axes concerned are no longer referenced (status flag "Homed" is set to FALSE).';
	16#4010: sMsg := '4010 parameter "Channel identifier not allowed" Either an unacceptable value (not 1...255) has been used, or a channel that does not exist in the system has been named.';
	16#4011: sMsg := '4011 parameter "Group identifier not allowed" Either an unacceptable value (not 1...255) has been used, or a group that does not exist in the system has been named.';
	16#4012: sMsg := '4012 parameter "Axis identifier not allowed" Either an unacceptable value (not 1...255) has been used, or an axis that does not exist in the system has been named.';
	16#4013: sMsg := '4013 parameter "Encoder identifier not allowed" Either an unacceptable value (not 1...255) has been used, or a encoder that does not exist in the system has been named.';
	16#4014: sMsg := '4014 parameter "Controller identifier not allowed" Either an unacceptable value (not 1...255) has been used, or a controller that does not exist in the system has been named.';
	16#4015: sMsg := '4015 parameter "Drive identifier not allowed" Either an unacceptable value (not 1...255) has been used, or a drive that does not exist in the system has been named.';
	16#4016: sMsg := '4016 parameter "Table identifier not allowed" Either an unacceptable value (not 1...255) has been used, or a table that does not exist in the system has been named.';
	16#4020: sMsg := '4020 internal "No process image" No PLC-axis interface during creation of an axis.';
	16#4021: sMsg := '4021 internal "No process image" No axis-PLC interface during creation of an axis.';
	16#4022: sMsg := '4022 internal "No process image" No encoder-I/O interface during creation of an axis.';
	16#4023: sMsg := '4023 internal "No process image" No I/O-encoder interface during creation of an axis.';
	16#4024: sMsg := '4024 internal "No process image" No drive-I/O interface during creation of an axis.';
	16#4025: sMsg := '4025 internal "No process image" No I/O-drive interface during creation of an axis.';
	16#4030: sMsg := '4030 internal "Coupling type not allowed" Unacceptable master/slave coupling type.';
	16#4031: sMsg := '4031 internal "Axis type not allowed" Unacceptable type specification during creation of an axis.';
	16#4040: sMsg := '4040 internal "Axis is incompatible" Axis is not suitable for the intended purpose. A high speed/low speed axis, for example, cannot function as a slave in an axis coupling.';
	16#4050: sMsg := '4050 internal "Channel not ready for operation" The channel is not complete, and is therefore not ready for operation. This is usually a consequence of problems at system start-up.';
	16#4051: sMsg := '4051 internal "Group not ready for operation" The group is not complete, and is therefore not ready for operation. This is usually a consequence of problems at system start-up.';
	16#4052: sMsg := '4052 internal "Axis not ready for operation" The axis is not complete, and is therefore not ready for operation. This is usually a consequence of problems at system start-up.';
	16#4060: sMsg := '4060 internal "Channel exists" The channel that is to be created already exists.';
	16#4061: sMsg := '4061 internal "Group exists" The group that is to be created already exists.';
	16#4062: sMsg := '4062 internal "Axis exists" The axis that is to be created already exists.';
	16#4063: sMsg := '4063 internal "Table exists" The table that is to be created already exists, resp. it is tried internally to use an already existing table id ( e.g. for the universal flying saw).';
	16#4070: sMsg := '4070 internal "Axis index not allowed" The location within the channel specified for an axis is not allowed.';
	16#4071: sMsg := '4071 internal "Axis index not allowed" The location within the group specified for an axis is not allowed.';
	16#4101: sMsg := '4101 internal "Group index not allowed" The location within the channel specified for an group is not allowed.';
	16#4102: sMsg := '4102 address "Null pointer" The pointer to the group is invalid. This is usually a consequence of an error at system start-up.';
	16#4103: sMsg := '4103 internal "No process image" It is not possible to exchange data with the PLC. Possible causes: n The channel does not have an interface (no interpreter present) n The connection to the PLC is faulty';
	16#4104: sMsg := '4104 parameter "M-function index not allowed" Unacceptable M-function (not 0...159) detected at the execution level.';
	16#4105: sMsg := '4105 memory "No memory" No more system memory is available. This is usually the result of another error.';
	16#4106: sMsg := '4106 internal "Not ready" The function is not presently available, because a similar function is already being processed. ';
	16#4107: sMsg := '4107 function "Function/command not supported" A requested function or command is not supported by the channel.';
	16#4108: sMsg := '4108 parameter "Invalid parameter while starting" Parameters to start the channel (TwinCAT-Start) are invalid. Typically there is an invalid memory size or channel type requested.';
	16#4109: sMsg := '4109 function "Channel function/command not executable" A channel function e.g. interpreter start is not executable because the channel is already busy, no program is loaded or in an error state.';
	16#410A: sMsg := '410A function "ItpGoAhead not executable" The requested command is not executable, because the interpreter is not executing a dekoder stop.';
	16#4110: sMsg := '4110 internal "Error opening a file" The specified file does not exist. Example: NC program unknown.';
	16#4111: sMsg := '4111 internal "Syntax error during loading" The NC has found a syntax error when loading an NC program.';
	16#4112: sMsg := '4112 internal "Syntax error during interpretation" The NC has found a syntax error when executing an NC program.';
	16#4113: sMsg := '4113 internal "Missing subroutine" The NC has found a missing subroutine while loading.';
	16#4114: sMsg := '4114 memory "Loading buffer of interpreter is too small" The capacity of the interpreter loading buffer has been exceeded.';
	16#4115: sMsg := '4115 internal „Symbolic” - reserved';
	16#4116: sMsg := '4116 internal „Symbolic” - reserved';
	16#4117: sMsg := '4117 internal „Subroutine incomplete” Header of subroutine is missing';
	16#4120: sMsg := '4120 internal "Divide by zero" The NC encountered a computation error during execution: division by 0.';
	16#4121: sMsg := '4121 internal "Invalid circle parameterisation" The NC encountered a computation error during execution: The specified circle cannot be calculated.';
	16#4122: sMsg := '4122 internal „Invalid FPU-Operation” The NC encountered an invalid FPU-Operation during exectuion. This error occurs e.g. by calculating the square root of a negative number.';
	16#4130: sMsg := '4130 internal "Stack overflow: subroutines" The NC encountered a stack overflow during execution: too many subroutine levels.';
	16#4131: sMsg := '4131 internal "Stack underflow: subroutines" The NC encountered a stack underflow during execution: too many subroutine return commands. Note: A main program must not end with a return command.';
	16#4132: sMsg := '4132 internal "Stack overflow: arithmetic unit" The NC encountered a stack overflow during execution: The calculation is too complex, or has not been correctly written.';
	16#4133: sMsg := '4133 internal "Stack underflow: arithmetic unit" The NC encountered a stack underflow during execution: The calculation is too complex, or has not been correctly written.';
	16#4140: sMsg := '4140 parameter "Register index not allowed" The NC encountered an unacceptable register index during execution: Either the program contains an unacceptable value (not R0...R999) or a pointer register contains an una…';
	16#4141: sMsg := '4141 parameter "Unacceptable G-function index" The NC has encountered an unacceptable G-function (not 0...159) during execution.';
	16#4142: sMsg := '4142 parameter "Unacceptable M-function index" The NC has encountered an unacceptable M-function (not 0...159) during execution.';
	16#4143: sMsg := '4143 parameter "Unacceptable extended address" The NC has encountered an unacceptable extended address (not 1...9) during execution.';
	16#4144: sMsg := '4144 parameter "Unacceptable index to the internal H-function" The NC has encountered an unacceptable internal H-function in the course of processing. This is usually a consequence of an error during loading.';
	16#4145: sMsg := '4145 parameter "Machine data value unacceptable" While processing instructions the NC has detected an impermissible value for the machine data (MDB) (not 0…7).';
	16#4150: sMsg := '4150 internal "Cannot change tool params here" The NC has encountered an unacceptable change of parameters for the tool compensation during execution. This error occured for instance by changing the tool radius and…';
	16#4151: sMsg := '4151 internal "Cannot calculate tool compensation" The NC has encountered an error by the calculation of the tool compensation';
	16#4152: sMsg := '4152 internal Tool compensation: The plane for the tool compensation cannot be changed here. This error occured for instance by changing the tool plane when the compensation is turned on or active.';
	16#4153: sMsg := '4153 internal Tool compensation: The D-Word is missing or invalid by turning on the tool compensation.';
	16#4154: sMsg := '4154 internal Tool compensation: The spezified tool radius is invalid because the value is less or equal zero.';
	16#4155: sMsg := '4155 internal Tool compensation: The tool radius cannot be changed here';
	16#4156: sMsg := '4156 internal Tool compensation: Collision Detection Table is full.';
	16#4157: sMsg := '4157 internal Tool compensation: Internal error while turning on the contour collision detection. ';
	16#4158: sMsg := '4158 internal Tool compensation: Internal error within the contour collision detection - update reversed geo failed.';
	16#4159: sMsg := '4159 internal Tool compensation: Unexpected combination of geometrie types by active contour collision detection.';
	16#415A: sMsg := '415A internal Tool compensation: Programmed inner circle is smaller than the cutter radius';
	16#415B: sMsg := '415B internal Tool compensation: Bottle neck detection recognized contour violation';
	16#415C: sMsg := '415C memory Table for corrected entries is full';
	16#415D: sMsg := '415D memory Input table for tangential following is full';
	16#415E: sMsg := '415E memory Executing table for tangential following is full';
	16#415F: sMsg := '415F internal Geometric entry for tangential following can not be calculated';
	16#4160: sMsg := '4160 internal reserved';
	16#4161: sMsg := '4161 internal reserved';
	16#4162: sMsg := '4162 internal The acutal active interpolation rules (g-code), zero-shifts, or rotation cannot be detected';
	16#4170: sMsg := '4170 internal "Error while loading: Invalid parameter" The NC has found an invalid parameter while loading an NC program.';
	16#4171: sMsg := '4171 internal "Invalid contour start position" The NC encountered a computation error during execution: The specified contour cannot be calculated because the initial position is not on the contour.';
	16#4200: sMsg := '4200 parameter "Group ID not allowed" The value for the group ID is not allowed, e.g. because it has already been assigned, is less than or equal to zero, or is greater than 255.';
	16#4201: sMsg := '4201 parameter "Group type not allowed" The value for the group type is unacceptable because it is not defined. Type 1: PTP group with slaves (servo) Type 5: DXD group with slaves (3D group) Type 6: High/low speed g…';
	16#4202: sMsg := '4202 internal "Master axis index not allowed" The value for the master axis index in an interpolating 3D group is not allowed, because, for instance, it has gone outside the value range. Index 0: X axis (first mast…';
	16#4203: sMsg := '4203 initialization "Slave axis index not allowed" (INTERNAL ERROR) . Index 0: First slave axis Index 1: Second slave axis Index 2: etc.';
	16#4204: sMsg := '4204 initialization "" (INTERNAL ERROR) GROUPERR_INTERNAL';
	16#4205: sMsg := '4205 parameter "Invalid cycle time for statement execution task (SAF)" The value of the cycle time for the NC block execution task (SAF 1/2) is not allowed, because it has passed outside the value range.';
	16#4206: sMsg := '4206 initialization "" GROUPERR_RANGE_MAXELEMENTSINAXIS';
	16#4207: sMsg := '4207 parameter "Invalid cycle time for the statement preparation task (SVB)" The value of the cycle time for the NC statement preparation task (SVB 1/2) is not allowed, because it has passed outside the value range.…';
	16#4208: sMsg := '4208 parameter "Single step mode not allowed" The flag for the activation or deactivation of single step mode is not allowed. Value 0: Passive (buffered operation) Value 1: Active (single-block operation)';
	16#4209: sMsg := '4209 parameter "Group deactivation not allowed" (INTERNAL ERROR) The flag for the deactivation or activation of the complete group is not allowed. Value 0: Group active Value 1: Group passive';
	16#420A: sMsg := '420A initialization "Statement execution state (SAF state) not allowed" (INTERNAL ERROR) The value for the state of the block execution state machine (SAF state) is not allowed. This error occurs on passing outside the r…';
	16#420B: sMsg := '420B address "Channel address" The group does not have a channel, or the channel address has not been initialised.';
	16#420C: sMsg := '420C address "Axis address (master axis)" The group does not have a master axis (or axes) or the axis address(es) has (have) not been initialised.';
	16#420D: sMsg := '420D address "Master axis address" A new master/slave coupling is to be inserted into the group, but there is no valid address for the leading master axis.';
	16#420E: sMsg := '420E address "Slave axis address" A master/slave coupling is to be inserted into the group, but there is no valid address for the slave axis.';
	16#420F: sMsg := '420F address "Slave set value generator address" A master/slave coupling is to be inserted into the group, but there is no valid address for the slave set value generator.';
	16#4210: sMsg := '4210 address "Encoder address" An axis in the group does not have an encoder, or the encoder address has not been initialised.';
	16#4211: sMsg := '4211 address "Controller address" An axis in the group does not have a controller, or the controller address has not been initialised.';
	16#4212: sMsg := '4212 address "Drive address" An axis in the group does not have a drive, or the drive address has not been initialised.';
	16#4213: sMsg := '4213 address "GROUPERR_ADDR_MASTERGENERATOR"';
	16#4214: sMsg := '4214 address "Axis interface NC to PLC address" Group/axis does not have an axis interface from the NC to the PLC, or the axis interface address has not been initialised.';
	16#4215: sMsg := '4215 address "Slave axis address" An existing master/slave coupling is to be removed from the group, but there is no valid address for the slave axis.';
	16#4216: sMsg := '4216 address „Table adress unknown“ The table, respectively the table ID, is unknown. This table is used for the master/slave coupling or for the characteristic curve.';
	16#4217: sMsg := '4217 address "NcControl address" The NcControl address has not been initialised.';
	16#4218: sMsg := '4218 initialization "Axis is blocked for commands while persistent NC data are queued" Axis is blocked for commands while waiting for valid IO data to accept the queued persistent NC data.';
	16#4219: sMsg := '4219 function "The scaling mode MASTER-AUTOOFFSET is invalid because no reference table was found". The used scaling mode MASTER-AUTOOFFSET is invalid in this context because an existing reference table is missing.…';
	16#421A: sMsg := '421A parameter "The master axis start position does not permit synchronisation" When a slave axis is being coupled on, the position of the master axis does not permit synchronisation at the given synchronisation pos…';
	16#421B: sMsg := '421B parameter "Slave coupling factor (gearing factor) of 0.0 is not allowed" A master/slave coupling with a gearing factor of 0.0 is being created. This value is not allowed, since it does not correspond to any pos…';
	16#421C: sMsg := '421C function "Insertion of master axis into group not allowed" A master axis is to be inserted into a group at a location that is already occupied by another master axis.';
	16#421D: sMsg := '421D function "Deletion of master axis from group not allowed" (INTERNAL ERROR) A master axis is to be removed from a location in a group that is not in fact occupied by master axis.';
	16#421E: sMsg := '421E function „Function/feature is not supported from the setpoint generator A function or feature is not supported from the setpoint generator (e.g. PTP master setpoint generator). This can be in general or only i…';
	16#421F: sMsg := '421F initialization "Group initialisation" Group has not been initialised. Although the group has been created, the rest of the initialisation has not been performed (1. Initialisation of group I/O, 2. Initialisation of …';
	16#4220: sMsg := '4220 monitoring "Group not ready / group not ready for new task" The group is being given a new task while it is still in the process of executing an existing task. This request is not allowed because it would interr…';
	16#4221: sMsg := '4221 monitoring "Requested set velocity is not allowed" The value requested for the set velocity of a positioning task is less than or equal to zero, larger than the "maximum velocity" ';
	16#4222: sMsg := '4222 monitoring "Requested target position is not allowed (master axis)" The requested value for the target position of a positioning task is not within the software end locations. location or larger than the maximum…';
	16#4223: sMsg := '4223 monitoring "No enable for controller and/or feed (Master axis)" The axis enables for the master axis needed for positioning are not present. This can involve the controller enable and/or the relevant, direction-…';
	16#4224: sMsg := '4224 monitoring "Movement smaller than one encoder increment" (INTERNAL ERROR) The distance that a group/axis is supposed to move is smaller than the physical significance of one encoder increment. In other words the…';
	16#4225: sMsg := '4225 monitoring "Drive not ready during axis start" During an axis start it is ascertained that the drive is not ready. The following are possible causes: - the drive is in failure state (hardware fault)';
	16#4226: sMsg := '4226 parameter "Invalid parameters of the emergency stop." The parameter of the E-Stop are invalid. Either the deceleration and the jerk are less than zero or one of the parameters is weaker than the corresponding p…';
	16#4227: sMsg := '4227 function "The setpoint generator is inactive such that no instructions are accepted."';
	16#4228: sMsg := '4228 monitoring „Requested traverse distance is not allowed“ The requested traverse distance or looping distance is smaller than the braking distance of the two/speed axis.';
	16#4229: sMsg := '4229 monitoring "Requested target position is not allowed (slave axis)" The value for the target position of a positioning task when calculated for the slave axis is not within the software end locations. ';
	16#422A: sMsg := '422A monitoring "No enable for controller and/or feed (slave axis)" The axis enables for one or more coupled slave axes needed for positioning are not present. This can involve the controller enable and/or the releva…';
	16#422B: sMsg := '422B parameter "The activation position (position threshold) is out of range of the actual positioning"';
	16#422C: sMsg := '422C monitoring The start or activation data of the external setpoint generation are not valid“ This may be caused through:';
	16#422D: sMsg := '422D function „Velocity is not constant“ For changing the dynamic parameter acceleration und deceleration the axis has to be in dynamic state without acceleration and deceleration (that means constant velocity)…';
	16#422E: sMsg := '422E parameter "Jerk less than or equal to 0.0 is not allowed" A value less than or equal to 0.0 for the jerk (PTP and CNC) is not allowed, since the jerk is by definition positive, and with a jerk of 0.0, division …';
	16#422F: sMsg := '422F parameter "Acceleration less than or equal to 0.0 is not allowed" A value less than or equal to 0.0 for the acceleration (PTP and CNC) is not allowed, since the acceleration is positive by definition, and an ac…';
	16#4230: sMsg := '4230 parameter "Absolute deceleration value less than or equal to 0.0 is not allowed" A value less than or equal to 0.0 for the absolute value of the deceleration (PTP and CNC) is not allowed';
	16#4231: sMsg := '4231 parameter "Set velocity less than or equal to 0.0 is not allowed" A value less than or equal to 0.0 or outside the range from 10-3 up to 10+10 for the set velocity (PTP and CNC) is not allowed';
	16#4232: sMsg := '4232 monitoring „Loss of precision when trying a positioning“ The positioning is so long in space or time that decimal parts loose there relevance LOSS_OF_PRECISION).';
	16#4233: sMsg := '4233 parameter "Cycle time less than or equal to 0.0 is not allowed" A value less than or equal to 0.0 for the cycle time (PTP and CNC) is not allowed, since the cycle time is by definition strictly positive, and wi…';
	16#4234: sMsg := '4234 internal "PTP data type <intasdouble> range exceeded" Such extreme parameters have been supplied for the start task, the override or the new target position that the internal data type loses its precision.';
	16#4235: sMsg := '4235 function "PTP LHL velocity profile cannot be generated" (INTERNAL ERROR) Such extreme parameters have been supplied for the start task, the override or the new target position that it is not possible to genera…';
	16#4236: sMsg := '4236 function "PTP HML velocity profile cannot be generated" (INTERNAL ERROR) Such extreme parameters have been supplied for the override or the new target position that it is not possible to generate a velocity pr…';
	16#4237: sMsg := '4237 address "Start data address is invalid" The address of the start data is invalid.';
	16#4238: sMsg := '4238 parameter "Velocity override (start override) is not allowed" The value for the velocity override is not allowed, because it is less than 0.0% or more than 100.0% (see axis interface PlcToNc). Here, 100.0 % cor…';
	16#4239: sMsg := '4239 parameter "Start type not allowed" The start type supplied does not exist.';
	16#423A: sMsg := '423A monitoring "Velocity overflow (overshoot in the velocity)" The new dynamic with the parameterized jerk is so weak that a velocity overflow will occur (overshoot in the velocity). The command is therefore not sup…';
	16#423B: sMsg := '423B parameter "Start parameter for the axis structure is invalid" External or internal parameters for the start structure for a positioning task are invalid. Thus, for instance, the scaling factor, the SAF cycle ti…';
	16#423C: sMsg := '423C parameter "Override generator initialisation parameter invalid" One of the override generator (re)initialisation parameters is invalid.';
	16#423D: sMsg := '423D monitoring "Slave axis has not set value generator" (INTERNAL ERROR) It is found that a slave axis within a group does not have a valid slave generator (set value generator). A slave axis and a slave set value g…';
	16#423E: sMsg := '423E function "Table is empty" Either the SVB table or the SAF table does not contain any entries.';
	16#423F: sMsg := '423F function "Table is full" The SVB table or the SAF table has no more free lines.';
	16#4240: sMsg := '4240 memory "No memory available" SVB memory allocation for dynamic entry in SAF table failed.';
	16#4241: sMsg := '4241 function "Table already contains an entry"(INTERNAL ERROR) SAF table entry abandoned, because, incorrectly, an entry already exists.';
	16#4242: sMsg := '4242 function "Stop is already active" The stop instruction is not forwarded, because it has already been activated.';
	16#4243: sMsg := '4243 function "Compensation has not been carried out over the full compensation section" The compensations start parameters do not permit compensation over the full section to be compensated. For this reason the co…';
	16#4244: sMsg := '4244 parameter "Start parameter address for the compensation invalid" (INTERNAL ERROR) Invalid address.';
	16#4245: sMsg := '4245 function "Compensation active" Start of compensation refused, because compensation is already active. ItS also possible that the M/S axes are NOT active moved. Therefore an execution OF the compensation is im…';
	16#4246: sMsg := '4246 function "Compensation not active" Stop of compensation refused, because compensation is not active.';
	16#4247: sMsg := '4247 function "Compensation type invalid" The type supplied for the section compensation is invalid. At the present time only compensation type 1 (trapezoidal velocity profile) is allowed.';
	16#4248: sMsg := '4248 function "Axis address for compensation invalid" (INTERNAL ERROR) The address of the master of slave axis on which the section compensation is to act is invalid. This is an internal error.';
	16#4249: sMsg := '4249 address "Invalid slave address" (INTERNAL ERROR) The slave address given for on-line coupling/decoupling is invalid.';
	16#424A: sMsg := '424A function "Coupling velocity invalid" The velocity of what is to become the master axis is 0, which means that on-line coupling is not possible.';
	16#424B: sMsg := '424B function "Coupling velocities not constant" The velocity of what is to become the master axis and the velocity of what is to become the slave axis are not constant, so that on-line coupling is not possible.';
	16#424C: sMsg := '424C parameter "Cycle time less than or equal to 0.0 is not allowed" A value less than or equal to 0.0 for the cycle time (Slave) is not allowed, since the cycle time is by definition strictly positive, and with a c…';
	16#424D: sMsg := '424D function "Decoupling task not allowed" The slave axis is of such a type (e.g. a table slave) or is in such a state (master velocity 0) that on-line decoupling is not possible.';
	16#424E: sMsg := '424E function "Function not allowed" The function cannot logically be executed, e.g. some commands are not possible and not allowed for slave axes.';
	16#424F: sMsg := '424F parameter "No valid table weighting has been set" The weighting factor of each table is 0, so that no table can be read.';
	16#4250: sMsg := '4250 function "Axis type, actual position type or end position type is not allowed" The start type for a positioning task in invalid. Valid start types are ABSOLUTE (1), RELATIVE (2), CONTINUOUS POSITIVE (3), CONTI…';
	16#4251: sMsg := '4251 function "Function not presently supported" An NC function has been activated that is currently not released for use, or which is not even implemented. This can be a command which is not possible or not allowe…';
	16#4252: sMsg := '4252 monitoring "State of state machine invalid" (INTERNAL ERROR) The state of an internal state machine is invalid. This is an internal error.';
	16#4253: sMsg := '4253 monitoring "Reference cam became free too soon" During the referencing process for an axis it is moved in the direction of the referencing cam, and is only stopped again when the cam signal is reached.';
	16#4254: sMsg := '4254 monitoring "Clearance monitoring between activation of the hardware latch and appearance of the sync pulse" When the clearance monitoring is active, a check is kept on whether the number of increments between ac…';
	16#4255: sMsg := '4255 memory "No memory available" The dynamic memory allocation for the set value generator, the SVB table or the SAF table has failed.';
	16#4256: sMsg := '4256 monitoring "The table slave axis has no active table" Although the table slave axis has tables, none of the tables is designated as active. If this occurs during the run time the whole master/slave group is stop…';
	16#4257: sMsg := '4257 function "Function not allowed" The requested function or the requested task is not logically allowed. An example for such an error message would be "set an actual position" for an absolute encoder (M3000, KL5…';
	16#4258: sMsg := '4258 function "Stopping compensation not allowed" It is not possible to stop the compensation, since compensation is already in the stopping phase.';
	16#4259: sMsg := '4259 function "Slave table is being used" The slave table cannot be activated, because it is currently being used.';
	16#425A: sMsg := '425A function "Master or slave axis is processing a job (e.g. positioning command) while coupling is requested" A master/slave coupling of a certain slave type (e.g. linear coupling) can not be executed. he master …';
	16#425B: sMsg := '425B parameter "Slave (start) parameter is incorrect" One of the slave start/coupling parameters is not allowed (Coupling factor is zero,t he master position scaling of an cam is zero, etc) .';
	16#425C: sMsg := '425C parameter "Slave type is incorrect" The slave type does not match up to the (SVB) start type.';
	16#425D: sMsg := '425D function "Axis stop is already active" The axis stop/Estop is not initiated, because the stop/estop is already active.';
	16#425E: sMsg := '425E function "Maximum number of tables per slavegenerator reached" The maximum number of tables per slave generator is reached (e.g. "MC_MultiCamIn" is limited to 4 tables).';
	16#425F: sMsg := '425F function "The scaling mode is invalid". The used scaling is invalid in this context. Either the mode is not defined or yet not implemented or however it cannot in this constellation be put into action.';
	16#4260: sMsg := '4260 monitoring "Controller enable" Controller enable for the axis or for a coupled slave axis is not present (see axis interface PlcToNc). This error occurs if the controller enable is withdrawn while an axis or a g…';
	16#4261: sMsg := '4261 function "Table not found" No table exists with the ID prescribed or the table ID is not unique.';
	16#4262: sMsg := '4262 function "Incorrect table type" The table referred to in the function is of the incorrect type.';
	16#4263: sMsg := '4263 function "Single step mode" This error occurs if single step mode is selected for a group or axis and a new task is requested while one of the individual tasks is still being processed.';
	16#4264: sMsg := '4264 function "Group task unknown (asynchronous table entry)" The group has received a task whose type or sub-type is unknown. Valid tasks can be single or multi-dimensional positioning tasks (Geo 1D, Geo 3D), refe…';
	16#4265: sMsg := '4265 function "Group function unknown (synchronous function)" The group has received a function whose type is unknown. Valid functions are "Reset", "Stop", "New end position", "Start/stop section compensation", "Se…';
	16#4266: sMsg := '4266 function "Group task for slave not allowed" Group tasks are usually only possible for master axes, not for slave axes. A slave axis only moves as an indirect result of a positioning task given to its associate…';
	16#4267: sMsg := '4267 function "Group function for slave not allowed" Group functions are in principle only possible for master axes, not for slave axes. The only exception is represented by the "Start/stop section compensation" fu…';
	16#4268: sMsg := '4268 function "GROUPERR_GROUPFUNC_NOMOTION"';
	16#4269: sMsg := '4269 parameter „Startposition=Setpoint Position“ Invalid position parameters.';
	16#426A: sMsg := '426A parameter „Parameters of the delay-denerator are invalid“ Invalid external/internal parameters of the delay generator (delay time, cycle time, tics).';
	16#426B: sMsg := '426B parameter „External parameters of the superimposed instruction are invalid“ Invalid external parameters of the superimposed functionality (acceleration, deceleration, velocity, process velocity, length).';
	16#426C: sMsg := '426C parameter "Invalid overridetype." The override type does not exist.';
	16#426D: sMsg := '426D function „Activation position under/overrun“ The requested activation position is located in the past of the master (e.g. when exchanging a cam table).';
	16#426E: sMsg := '426E function „Activation impossible: Master is standing“ The required activation of the correction is impossible since the master axis is not moving. A synchronisation is not possible, because the master axis stan…';
	16#426F: sMsg := '426F function „Activation mode not possible“ The requested activation mode is not possible when the slave axis is moving (otherwise the slave velocity would jump to zero).';
	16#4270: sMsg := '4270 parameter "Start parameter for the compensation is invalid" One of the dynamic parameters for the compensation is invalid (necessary condition): Acceleration (>0) Deceleration (>0) Process velocity (>0)';
	16#4271: sMsg := '4271 parameter "Start parameter for the compensation is invalid" Velocity camber is negative.';
	16#4272: sMsg := '4272 parameter "Start parameter for the compensation is invalid" The section on which the compensation is to occur is not positive.';
	16#4273: sMsg := '4273 monitoring „Target position under/overrun“ (INTERNAL ERROR) The position (calculated from the modulo-target-position) where the axis should stand at end of oriented stop has been run over.';
	16#4274: sMsg := '4274 monitoring „Target position will be under/overrun“ (INTERNAL ERROR) The position (calculated from the modulo-target-position) where the axis should stand at end of oriented stop is too near and will be run over.…';
	16#4276: sMsg := '4276 monitoring "GROUPERR_GUIDERSTARTDATA"';
	16#4277: sMsg := '4277 monitoring „Dynamic parameters not permitted“ (INTERNAL ERROR) The dynamic parameters resulting from internal calculation like acceleration, deceleration and jerk are not permitted.';
	16#4279: sMsg := '4279 monitoring "GROUPERR_GUIDEROVERRUN"';
	16#427A: sMsg := '427A monitoring "GROUPERR_GUIDERLOOKAHEAD"';
	16#427B: sMsg := '427B monitoring "GROUPERR_GUIDERLOOKAHEADEND"';
	16#427C: sMsg := '427C monitoring "GROUPERR_GUIDERLOOKAHEADREQU"';
	16#427D: sMsg := '427D monitoring "GROUPERR_GUIDERMODE"';
	16#427E: sMsg := '427E monitoring „A requested motion command could not be realized (BISECTION)“ A requested motion command could not be realized using the requested parameters. The command has been executed best possible and this mes…';
	16#427F: sMsg := '427F monitoring „The new target position either has been overrun or will be overrun“ The new target position either has been overrun or will be overrun, since until there it is impossible to stop. A internal stop com…';
	16#4280: sMsg := '4280 monitoring "Group not ready / group not ready for new task" (INTERNAL ERROR / INFORMATION) The group is being given a new task while it is still in the process of executing an existing task. This request is not …';
	16#4281: sMsg := '4281 parameter "The parameters of the oriented stop (O-Stop) are not admitted." The modulo-target position should not be smaller than zero and not larger or equal than the encoder mod-period ( e.g. in the interval […';
	16#4282: sMsg := '4282 monitoring "The modulo target position of the modulo-start is invalid" The modulo target position is outside of the valid parameter range. So the position value should not be smaller than zero and not greater or…';
	16#4283: sMsg := '4283 parameter "The online change activation mode is invalid". The activation can be used with online scaling or with online modification of motion function. The used activation is invalid in this context……';
	16#4284: sMsg := '4284 parameter "The parameterized jerk rate is not permitted". The jerk rate is smaller than the minimum jerk rate. The minimum value for jerk rate is 1.0 (e.g. mm/s^3).';
	16#4285: sMsg := '4285 parameter "The parameterized acceleration or deceleration is not permitted". The parameterized acceleration or deceleration is lower than the permitted minimum acceleration. The value for minimum acceleration i…';
	16#4286: sMsg := '4286 parameter "The parameterized velocity is not permitted". The parameterized target velocity is lower than the minimum velocity (but the value zero is permitted). The value for minimum velocity is calculated from…';
	16#4287: sMsg := '4287 monitoring "A activation cannot be executed due to a pending activation" A activation e.g. "CamIn", "CamScaling" or "WriteMotionFunction" cannot be executed due to a pending activation (e.g. "CamIn", "CamScaling…';
	16#4288: sMsg := '4288 monitoring „Illegal combination of different cycle times within an axis group“ A logical axis group includes elements (axes) with different cycle times for a common setpoint generator and I/O-execution, resp. Th…';
	16#4289: sMsg := '4289 monitoring "Illegal motion reversal" Due to the actual dynamical state a motion reversal will happen. To avoid this motion reversal the axis command is not performed and the previous system state restored.';
	16#428A: sMsg := '428A monitoring „Illegal moment for an axis command because there is an old axis command with activation position still active“ The moment for the command is illegal because there is still an old command with activat…';
	16#428B: sMsg := '428B monitoring "Error in the stop-calculation routine" (INTERNAL ERROR) Due to an internal error in the stop-calculation routine the current commando cannot be performed. The previous system state is restored.';
	16#428C: sMsg := '428C monitoring "A command with activation position cannot fully be performed because the remaining path is too short"';
	16#428D: sMsg := '428D monitoring "Illegal decoupletype when decoupling a slave axis" The decouple and restart command contains an invalid decouple type.';
	16#428E: sMsg := '428E monitoring "Illegal target velocity when decoupling a slave axis" The decouple and restart command contains an illegal target velocity [1 < V <Vmax].';
	16#428F: sMsg := '428F monitoring "The command new dynamic parameter cannot be performed since this would require a new target velocity" ';
	16#4290: sMsg := '4290 monitoring „A command with activation position cannot be performed becaus the axis is already in the brake phase“';
	16#4291: sMsg := '4291 monitoring „Decouple routine of slave axis doesnt return a valid solution“';
	16#4292: sMsg := '4292 monitoring „Command not be executed because the command buffer is full filled“';
	16#4293: sMsg := '4293 internal „Command is rejected due to an internal error in the Look Ahead“ (INTERNAL ERROR)';
	16#4294: sMsg := '4294 monitoring „Command is rejected because the segment target velocity is not realized“';
	16#4295: sMsg := '4295 monitoring „Successive commands have the same final position“';
	16#4296: sMsg := '4296 monitoring „Logical positioning direction is inconsistent with the direction of the buffer command“';
	16#4297: sMsg := '4297 monitoring „Command is rejected because the remaining positioning length is to small“';
	16#429C: sMsg := '429C monitoring „Reference cam is not found“ During the referencing process for an axis it is moved in the direction of the referencing cam. This reference cam, however, was not found as expected (=> leads to the abo…';
	16#429D: sMsg := '429D monitoring "Reference cam became not free" During the referencing process for an axis it is moved in the direction of the referencing cam, and is only stopped again when the cam signal is reached. After the axis…';
	16#429E: sMsg := '429E monitoring “IO sync pulse was not found (only when using hardware latch)”. If the hardware latch is activated, a sync pulse (zero pulse) is expected to be found and a sync event triggered following the expiry of…';
	16#42A0: sMsg := '42A0 internal "Group/axis consequential error" Consequential error resulting from another causative error related to another axis within the group. Group/axis consequential errors can occur in relation to master/sl…';
	16#42A1: sMsg := '42A1 parameter "Velocity reduction factor for C0/C1 transition is not allowed" A C0 transition describes two geometries which, while they are themselves continuous, no not have either continuous first or second diff…';
	16#42A2: sMsg := '42A2 parameter "Critical angle at segment transition not allowed"';
	16#42A3: sMsg := '42A3 parameter "Radius of the tolerance sphere" is in an invalid range ';
	16#42A4: sMsg := '42A4 parameter Not implemented.';
	16#42A5: sMsg := '42A5 parameter "Start type"';
	16#42A6: sMsg := '42A6 parameter Not implemented.';
	16#42A7: sMsg := '42A7 parameter "Blending" with given parameters not possible';
	16#42A8: sMsg := '42A8 parameter Not implemented.';
	16#42A9: sMsg := '42A9 parameter "Curve velocity reduction method not allowed" (INTERNAL ERROR) The curve velocity reduction method does not exist.';
	16#42AA: sMsg := '42AA parameter "Minimum velocity not allowed" The minimum velocity that has been entered is less than 0.0.';
	16#42AB: sMsg := '42AB parameter "Power function input not allowed" (INTERNAL ERROR) The input parameters in the power_() function lead to an FPU exception.';
	16#42AC: sMsg := '42AC parameter "Dynamic change parameter not allowed" A parameter that controls alterations to the dynamics is invalid. parameters: 1. Absolute motion dynamics change: All parameters must be strictly positive. 2. Re…';
	16#42AD: sMsg := '42AD memory "Memory allocation error" (INTERNAL ERROR)';
	16#42AE: sMsg := '42AE function "The calculated end position differs from the end position in the nc instruction (internal error)."';
	16#42AF: sMsg := '42AF parameter "Calculate remaining chord length"';
	16#42B0: sMsg := '42B0 function "Set value generator SVB active" Starting the set value generator (SVB, SAF) has been refused, since the SVB task is already active.';
	16#42B1: sMsg := '42B1 parameter "SVB parameter not allowed" (INTERNAL ERROR) A parameter related to the internal structure of the set value generator (SVB) results in logical errors and/or to an FPU exception. Affects these paramete…';
	16#42B2: sMsg := '42B2 parameter "Velocity reduction factor not allowed" A parameter that controls reduction of the velocity at segment transitions is invalid. Parameters: 1. Transitions with continuous first differential: VeloVertex…';
	16#42B3: sMsg := '42B3 parameter "Helix is a circle" The helix has degenerated to a circle, and should be entered as such.';
	16#42B4: sMsg := '42B4 parameter "Helix is a straight line" The helix has degenerated to a straight line, and should be entered as such.';
	16#42B5: sMsg := '42B5 parameter "Guider parameter not allowed" One of the guiders parameters leads to logical errors and/or to an FPU exception.';
	16#42B6: sMsg := '42B6 address "Invalid segment address" (INTERNAL ERROR) The geometry segment does not have a valid geometry structure address or does not have a valid dynamic structure address.';
	16#42B7: sMsg := '42B7 parameter "Unparametrised generator" (INTERNAL ERROR) The SVB generator is not yet parameterised and is therefore unable to operate.';
	16#42B8: sMsg := '42B8 address "Unparametrised table" (INTERNAL ERROR) The table has no information concerning the address of the corresponding dynamic generator.';
	16#42BA: sMsg := '42BA internal "The calculation of the arc length of the smoothed path failed (internal error)."';
	16#42BB: sMsg := '42BB parameter "The radius of the tolerance ball is too small (smaller than 0.1 mm)."';
	16#42BC: sMsg := '42BC internal Error while calculating DXD-Software-Limitswitches (internal error))';
	16#42BD: sMsg := '42BD function "NC-Block violates software limit switches of the group" At least one path axis with active software limit monitoring has violated the limit switches Therefore the geometric entry is denied with an er…';
	16#42BE: sMsg := '42BE parameter "GROUPERR_DXD_SOFTENDCHECK"';
	16#42BF: sMsg := '42BF parameter "GROUPERR_DXD_RTTG_VELOREFERENCE"';
	16#42C0: sMsg := '42C0 internal "Interpolating group contains axes of an incorrect axis type" An interpolating 3D group may only contain continuously guided axes of axis type 1 (SERVO).';
	16#42C1: sMsg := '42C1 internal "Scalar product can not be calculated" The length of one of the given vectors is 0.0.';
	16#42C2: sMsg := '42C2 internal "Inverse cosine can not be calculated" The length of one of the given vectors is 0.0.';
	16#42C3: sMsg := '42C3 parameter "Invalid table entry type" The given table entry type is unknown.';
	16#42C4: sMsg := '42C4 parameter "Invalid DIN66025 information type" (INTERNAL ERROR) The given DIN66025 information type is unknown. Known types: G0, G1, G2, G3, G17, G18, G19.';
	16#42C5: sMsg := '42C5 parameter "Invalid dimension" (INTERNAL ERROR) The CNC dimension is unknown. Known dimensions: 1, 2, 3. Or: The CNC dimension is invalid for the given geometrical object. For a circle the dimension must be 2 or…';
	16#42C6: sMsg := '42C6 parameter "Geometrical object is not a straight line" The given object, interpreted as a straight line, has a length of 0.0.';
	16#42C7: sMsg := '42C7 parameter "Geometrical object is not a circle" Interpreted as a circular arc, the given object has a length of 0.0, or an angle of 0.0 or a radius of 0.0.';
	16#42C8: sMsg := '42C8 parameter "Geometrical object is not a helix" Interpreted as a circular arc, the given object has a length of 0.0, or an angle of 0.0, or a radius of 0.0. or a height of 0.0.';
	16#42C9: sMsg := '42C9 parameter "Set velocity less than or equal to 0.0 is invalid" A value less than or equal to 0.0 for the set velocity (CNC) is not allowed, since the set velocity is positive by definition, and a set velocity of…';
	16#42CA: sMsg := '42CA address "Address for look-ahead invalid" (INTERNAL ERROR) The address supplied for the look-ahead is invalid.';
	16#42CB: sMsg := '42CB function "Set value generator SAF active" Starting the set value generator (SAF) has been refused, since the SAF task is already active.';
	16#42CC: sMsg := '42CC function "CNC set value generation not active" Stop or change of override refused, because the set value generation is not active.';
	16#42CD: sMsg := '42CD function "CNC set value generation in the stop phase" Stop or change of override refused, because the set value generation is in the stop phase.';
	16#42CE: sMsg := '42CE parameter "Override not allowed" An override of less than 0.0% or more than 100.0% is invalid.';
	16#42CF: sMsg := '42CF address "Invalid table address" (INTERNAL ERROR) The table address given for the initialisation of the set value generator is invalid, or no valid logger connection (report file) is present.';
	16#42D0: sMsg := '42D0 parameter "Invalid table entry type" The given table entry type is unknown.';
	16#42D1: sMsg := '42D1 memory "Memory allocation failed" Memory allocation for the table has failed.';
	16#42D2: sMsg := '42D2 memory "Memory allocation failed" Memory allocation for the filter has failed.';
	16#42D3: sMsg := '42D3 parameter "Invalid parameter" Filter parameter is not allowed.';
	16#42D4: sMsg := '42D4 function "Delete Distance To Go failed" Delete Distance to go (only interpolation) failed. This error occured, if e.g. the command DelDTG was not programmed in the actual movement of the nc program.';
	16#42D5: sMsg := '42D5 internal "The setpoint generator of the fying saw generates incompatible values (internal error)"';
	16#42D6: sMsg := '42D6 parameter "Axis will be stopped since otherwise it will overrun its target position (old PTP setpoint generator)" If, for example, in case of a slave to master transformation for the new master a target positio…';
	16#42D7: sMsg := '42D7 function "Internal error in the transformation from slave to master."';
	16#42D8: sMsg := '42D8 function "Wrong direction in the transformation of slave to master."';
	16#42DA: sMsg := '42DA parameter "Parameter of Motion Function (MF) table incorrect" The parameter of the Motion Function (MF) are incorrect. This may refer to the first time created data set or to online changed data.';
	16#42DB: sMsg := '42DB parameter "Parameter of Motion Function (MF) table invalid" The parameter of the Motion Function (MF) are invalid. This may refer to the first time created data set or to online changed data.';
	16#42DC: sMsg := '42DC monitoring "Internal error by using Motion Function (MF)" An internal error occurs by using the Function (MF). This error can not be solved by the user. Plaese ask the TwinCAT Support.';
	16#42DD: sMsg := '42DD function "Axis coupling with synchronization generator declined because of incorrect axis dynamic values" The axis coupling with the synchronization generator has been declined, because one of the slave dynami…';
	16#42DE: sMsg := '42DE function "Coupling conditions of synchronization generator incorrect"';
	16#42DF: sMsg := '42DF monitoring "Moving profile of synchronization generator declines dynamic limit of slave axis or required characterstic of profile" One of the parameterized checks has recognized an overstepping of the dynamic li…';
	16#42E0: sMsg := '42E0 parameter "Invalid parameter" The encoder generator parameter is not allowed.';
	16#42E1: sMsg := '42E1 parameter "Invalid parameter" The external (Fifo) generator parameter is not allowed.';
	16#42E2: sMsg := '42E2 function "External generator is active" The external generator cannot be started, as it is already active.';
	16#42E3: sMsg := '42E3 function "External generator is not active" The external generator cannot be stopped, as it is not active.';
	16#42E4: sMsg := '42E4 function "NC-Block with auxiliary axis violates software limit switches of the group" At least one auxiliary axis with active software limit monitoring has violated the limit switches Therefore the geometric e…';
	16#42E5: sMsg := '42E5 function "NC-Block type Bezier spline curve contains a cusp (singularity)" The Bezier spline curve contain a cusp, i.e. at a certain interior point both the curvature and the modulus of the velocity tend to 0 …';
	16#42E7: sMsg := '42E7 parameter „Value for dead time compensation not allowed“ The value for the dead time compensation in seconds for a slave coupling to an encoder axis (virtual axis) is not allowed.';
	16#42E8: sMsg := '42E8 parameter "GROUPERR_RANGE_NOMOTIONWINDOW"';
	16#42E9: sMsg := '42E9 parameter "GROUPERR_RANGE_NOMOTIONFILTERTIME"';
	16#42EA: sMsg := '42EA parameter "GROUPERR_RANGE_TIMEUNITFIFO"';
	16#42EB: sMsg := '42EB parameter "GROUPERR_RANGE_OVERRIDETYPE"';
	16#42EC: sMsg := '42EC parameter "GROUPERR_RANGE_OVERRIDECHANGETIME"';
	16#42ED: sMsg := '42ED parameter "GROUPERR_FIFO_INVALIDDIMENSION"';
	16#42EE: sMsg := '42EE address "GROUPERR_ADDR_FIFOTABLE"';
	16#42EF: sMsg := '42EF monitoring "Axis is locked for motion commands because a stop command is still active" The axis/group is locked for motion commands because a stop command is still active. The axis can be released by calling MC_…';
	16#42F0: sMsg := '42F0 parameter "Invalid number of auxiliary axes" The local number of auxiliary axes does not tally with the global number of auxiliary axes.';
	16#42F1: sMsg := '42F1 parameter "Invalid reduction parameter for auxiliary axes" The velocity reduction parameters for the auxiliary axes are inconsistent.';
	16#42F2: sMsg := '42F2 parameter "Invalid dynamic parameter for auxiliary axes" The dynamic parameters for the auxiliary axes are inconsistent.';
	16#42F3: sMsg := '42F3 parameter "Invalid coupling parameter for auxiliary axes" The coupling parameters for the auxiliary axes are inconsistent.';
	16#42F4: sMsg := '42F4 parameter "Invalid auxiliary axis entry" The auxiliary axis entry is empty (no axis motion).';
	16#42F6: sMsg := '42F6 parameter "Invalid parameter" The limit for velocity reduction of the auxiliary axes is invalid. It has to be in the interval 0..1.0';
	16#42FF: sMsg := '42FF monitoring "GROUPERR_HYMMEN_WATCHDOG"';
	16#4300: sMsg := '4300 parameter "Axis ID not allowed" The value for the axis ID is not allowed, e.g. because it has already been assigned, is less than or equal to zero, is greater than 255, or does not exist in the current configur…';
	16#4301: sMsg := '4301 parameter "Axis type not allowed" The value for the axis type is unacceptable because it is not defined. Type 1: Servo Type 2: High/low speed Type 3: Stepper motor';
	16#4306: sMsg := '4306 parameter "Slow manual velocity not allowed" The value for the slow manual velocity is not allowed.';
	16#4307: sMsg := '4307 parameter "Fast manual velocity not allowed" The value for the fast manual velocity is not allowed.';
	16#4308: sMsg := '4308 parameter "High speed not allowed" The value for the high speed is not allowed.';
	16#4309: sMsg := '4309 parameter "Acceleration not allowed" The value for the axis acceleration is not allowed.';
	16#430A: sMsg := '430A parameter "Deceleration not allowed" The value for the axis deceleration is not allowed.';
	16#430B: sMsg := '430B parameter "Jerk not allowed" The value for the axis jerk is not allowed.';
	16#430C: sMsg := '430C parameter "Delay time between position and velocity is not allowed" The value for the delay time between position and velocity ("idle time compensation") is not allowed.';
	16#430D: sMsg := '430D parameter „Override-Type not allowed” The value for the velocity override type is not allowed. Type 1: With respect to the internal reduced velocity (default value) Type 2: With respect to the original external…';
	16#430E: sMsg := '430E parameter "NCI: Velo-Jump-Factor not allowed"';
	16#430F: sMsg := '430F parameter "NCI: Radius of tolerance sphere for the auxiliary axes is invalid"';
	16#4310: sMsg := '4310 parameter "NCI: Value for maximum deviation for the auxiliary axes is invalid"';
	16#4312: sMsg := '4312 parameter "Referencing velocity in direction of cam not allowed" The value for the referencing velocity in the direction of the referencing cam is not allowed.';
	16#4313: sMsg := '4313 parameter "Referencing velocity in sync direction not allowed" The value for the referencing velocity in the direction of the sync pulse (zero track) is not allowed.';
	16#4314: sMsg := '4314 parameter "Pulse width in positive direction not allowed" The value for the pulse width in the positive direction is not allowed (pulsed operation). The use of the pulse width for positioning is chosen implicit…';
	16#4315: sMsg := '4315 parameter "Pulse width in negative direction not allowed" The value for the pulse width in the negative direction is not allowed (pulsed operation). The use of the pulse width for positioning is chosen implicit…';
	16#4316: sMsg := '4316 parameter "Pulse time in positive direction not allowed" The value for the pulse width in the positive direction is not allowed (pulsed operation).';
	16#4317: sMsg := '4317 parameter "Pulse time in negative direction not allowed" The value for the pulse width in the negative direction is not allowed (pulsed operation).';
	16#4318: sMsg := '4318 parameter "Creep distance in positive direction not allowed" The value for the creep distance in the positive direction is not allowed.';
	16#4319: sMsg := '4319 parameter "Creep distance in negative direction not allowed" The value for the creep distance in the negative direction is not allowed.';
	16#431A: sMsg := '431A parameter "Braking distance in positive direction not allowed" The value for the braking distance in the positive direction is not allowed.';
	16#431B: sMsg := '431B parameter "Braking distance in negative direction not allowed" The value for the braking distance in the negative direction is not allowed.';
	16#431C: sMsg := '431C parameter "Braking time in positive direction not allowed" The value for the braking time in the positive direction is not allowed.';
	16#431D: sMsg := '431D parameter "Braking time in negative direction not allowed" The value for the braking time in the negative direction is not allowed.';
	16#431E: sMsg := '431E parameter "Switching time from high to low speed not allowed" The value for the time to switch from high to low speed is not allowed.';
	16#431F: sMsg := '431F parameter "Creep distance for stop not allowed" The value for the creep distance for an explicit stop is not allowed.';
	16#4320: sMsg := '4320 parameter "Motion monitoring not allowed" The value for the activation of the motion monitoring is not allowed.';
	16#4321: sMsg := '4321 parameter "Position window monitoring not allowed" The value for the activation of the position window monitoring is not allowed.';
	16#4322: sMsg := '4322 parameter "Target window monitoring not allowed" The value for the activation of target window monitoring is not allowed.';
	16#4323: sMsg := '4323 parameter "Loop not allowed" The value for the activation of loop movement is not allowed.';
	16#4324: sMsg := '4324 parameter "Motion monitoring time not allowed" The value for the motion monitoring time is not allowed.';
	16#4325: sMsg := '4325 parameter "Target window range not allowed" The value for the target window is not allowed.';
	16#4326: sMsg := '4326 parameter "Position window range not allowed" The value for the position window is not allowed.';
	16#4327: sMsg := '4327 parameter "Position window monitoring time not allowed" The value for the position window monitoring time is not allowed.';
	16#4328: sMsg := '4328 parameter "Loop movement not allowed" The value for the loop movement is not allowed.';
	16#4329: sMsg := '4329 parameter "Axis cycle time not allowed" The value for the axis cycle time is not allowed.';
	16#432A: sMsg := '432A parameter "Stepper motor operating mode not allowed" The value for the stepper motor operating mode is not allowed.';
	16#432B: sMsg := '432B parameter "Displacement per stepper motor step not allowed" The value for the displacement associated with one step of the stepper motor is not allowed (step scaling). Value range: [0.000001, 1000.0] Unit: e.g.…';
	16#432C: sMsg := '432C parameter "Minimum speed for stepper motor set value profile not allowed" The value for the minimum speed of the stepper motor speed profile is not allowed.';
